	VAR robtarget OpenholeUD_1373 := [[450.39, 0.9, 181.06], [-0.062156, 0.70437, 0.703684, -0.06949], [0,0,0,0], [9E9, 9E9, 9E9, 9E9, 9E9, 9E9]];
	VAR robtarget OpenholeUD_1374 := [[446.46, 0.9, 181.82], [-0.075448, 0.70307, 0.704874, -0.056152], [0,0,0,0], [9E9, 9E9, 9E9, 9E9, 9E9, 9E9]];
	VAR robtarget OpenholeUD_1375 := [[442.53, 0.9, 182.57], [-0.088597, 0.701534, 0.705814, -0.042733], [0,0,0,0], [9E9, 9E9, 9E9, 9E9, 9E9, 9E9]];
	VAR robtarget OpenholeUD_1376 := [[438.6, 0.9, 183.32], [-0.101564, 0.699775, 0.7065, -0.029277], [0,0,0,0], [9E9, 9E9, 9E9, 9E9, 9E9, 9E9]];
	VAR robtarget OpenholeUD_1377 := [[434.67, 0.9, 184.08], [-0.114312, 0.697806, 0.70693, -0.015828], [0,0,0,0], [9E9, 9E9, 9E9, 9E9, 9E9, 9E9]];
	VAR robtarget OpenholeUD_1378 := [[430.74, 0.9, 184.83], [-0.126806, 0.695644, 0.707103, -0.002428], [0,0,0,0], [9E9, 9E9, 9E9, 9E9, 9E9, 9E9]];
	VAR robtarget OpenholeUD_1379 := [[426.82, 0.9, 185.59], [-0.139016, 0.693307, 0.707023, 0.010881], [0,0,0,0], [9E9, 9E9, 9E9, 9E9, 9E9, 9E9]];
	VAR robtarget OpenholeUD_1380 := [[422.89, 0.9, 186.34], [-0.150917, 0.690814, 0.706697, 0.024059], [0,0,0,0], [9E9, 9E9, 9E9, 9E9, 9E9, 9E9]];
	VAR robtarget OpenholeUD_1381 := [[418.96, 0.9, 187.09], [-0.162486, 0.688185, 0.706134, 0.03707], [0,0,0,0], [9E9, 9E9, 9E9, 9E9, 9E9, 9E9]];
	VAR robtarget OpenholeUD_1382 := [[415.03, 0.9, 187.85], [-0.173706, 0.685439, 0.705345, 0.049878], [0,0,0,0], [9E9, 9E9, 9E9, 9E9, 9E9, 9E9]];
	VAR robtarget OpenholeUD_1383 := [[411.1, 0.9, 188.6], [-0.184564, 0.682595, 0.704343, 0.062455], [0,0,0,0], [9E9, 9E9, 9E9, 9E9, 9E9, 9E9]];
	VAR robtarget OpenholeUD_1384 := [[407.17, 0.9, 189.35], [-0.195051, 0.679673, 0.703142, 0.074774], [0,0,0,0], [9E9, 9E9, 9E9, 9E9, 9E9, 9E9]];
	VAR robtarget OpenholeUD_1385 := [[403.25, 0.9, 190.11], [-0.205161, 0.67669, 0.701758, 0.086812], [0,0,0,0], [9E9, 9E9, 9E9, 9E9, 9E9, 9E9]];
	VAR robtarget OpenholeUD_1386 := [[399.32, 0.9, 190.86], [-0.214892, 0.673663, 0.700205, 0.098551], [0,0,0,0], [9E9, 9E9, 9E9, 9E9, 9E9, 9E9]];
	VAR robtarget OpenholeUD_1387 := [[395.39, 0.9, 191.62], [-0.224244, 0.670608, 0.698502, 0.109975], [0,0,0,0], [9E9, 9E9, 9E9, 9E9, 9E9, 9E9]];
	VAR robtarget OpenholeUD_1388 := [[389.38, 0.9, 192.77], [-0.237824, 0.665913, 0.695643, 0.126812], [0,0,0,0], [9E9, 9E9, 9E9, 9E9, 9E9, 9E9]];
	VAR robtarget OpenholeUD_1389 := [[385.38, 0.9, 192.78], [-0.183051, 0.683002, 0.683002, 0.183051], [0,0,0,0], [9E9, 9E9, 9E9, 9E9, 9E9, 9E9]];
	VAR robtarget OpenholeUD_1390 := [[381.38, 0.9, 192.79], [-0.183051, 0.683002, 0.683002, 0.183051], [0,0,0,0], [9E9, 9E9, 9E9, 9E9, 9E9, 9E9]];
	VAR robtarget OpenholeUD_1391 := [[377.38, 0.9, 192.81], [-0.183051, 0.683002, 0.683002, 0.183051], [0,0,0,0], [9E9, 9E9, 9E9, 9E9, 9E9, 9E9]];
	VAR robtarget OpenholeUD_1392 := [[373.38, 0.9, 192.82], [-0.183051, 0.683002, 0.683002, 0.183051], [0,0,0,0], [9E9, 9E9, 9E9, 9E9, 9E9, 9E9]];
	VAR robtarget OpenholeUD_1393 := [[369.38, 0.9, 192.83], [-0.183051, 0.683002, 0.683002, 0.183051], [0,0,0,0], [9E9, 9E9, 9E9, 9E9, 9E9, 9E9]];
	VAR robtarget OpenholeUD_1394 := [[369.38, 0.9, 192.83], [-0.183051, 0.683002, 0.683002, 0.183051], [0,0,0,0], [9E9, 9E9, 9E9, 9E9, 9E9, 9E9]];
	VAR robtarget OpenholeUD_1395 := [[369.38, 0.9, 192.95], [-0.183051, 0.683002, 0.683002, 0.183051], [0,0,0,0], [9E9, 9E9, 9E9, 9E9, 9E9, 9E9]];
	VAR robtarget OpenholeUD_1396 := [[373.38, 0.9, 192.94], [-0.183051, 0.683002, 0.683002, 0.183051], [0,0,0,0], [9E9, 9E9, 9E9, 9E9, 9E9, 9E9]];
	VAR robtarget OpenholeUD_1397 := [[377.38, 0.9, 192.93], [-0.183051, 0.683002, 0.683002, 0.183051], [0,0,0,0], [9E9, 9E9, 9E9, 9E9, 9E9, 9E9]];
	VAR robtarget OpenholeUD_1398 := [[381.38, 0.9, 192.91], [-0.183051, 0.683002, 0.683002, 0.183051], [0,0,0,0], [9E9, 9E9, 9E9, 9E9, 9E9, 9E9]];
	VAR robtarget OpenholeUD_1399 := [[385.38, 0.9, 192.9], [-0.183051, 0.683002, 0.683002, 0.183051], [0,0,0,0], [9E9, 9E9, 9E9, 9E9, 9E9, 9E9]];
	VAR robtarget OpenholeUD_1400 := [[389.38, 0.9, 192.89], [-0.237996, 0.665851, 0.695661, 0.126714], [0,0,0,0], [9E9, 9E9, 9E9, 9E9, 9E9, 9E9]];
	VAR robtarget OpenholeUD_1401 := [[393.31, 0.9, 192.14], [-0.229215, 0.668925, 0.697561, 0.115797], [0,0,0,0], [9E9, 9E9, 9E9, 9E9, 9E9, 9E9]];
	VAR robtarget OpenholeUD_1402 := [[397.24, 0.9, 191.38], [-0.220061, 0.671992, 0.699335, 0.10455], [0,0,0,0], [9E9, 9E9, 9E9, 9E9, 9E9, 9E9]];
	VAR robtarget OpenholeUD_1403 := [[401.17, 0.9, 190.63], [-0.210529, 0.675039, 0.700967, 0.092984], [0,0,0,0], [9E9, 9E9, 9E9, 9E9, 9E9, 9E9]];
	VAR robtarget OpenholeUD_1404 := [[405.1, 0.9, 189.87], [-0.200618, 0.678051, 0.702439, 0.08111], [0,0,0,0], [9E9, 9E9, 9E9, 9E9, 9E9, 9E9]];
	VAR robtarget OpenholeUD_1405 := [[409.02, 0.9, 189.12], [-0.190327, 0.681011, 0.703737, 0.068947], [0,0,0,0], [9E9, 9E9, 9E9, 9E9, 9E9, 9E9]];
	VAR robtarget OpenholeUD_1406 := [[412.95, 0.9, 188.37], [-0.17966, 0.683902, 0.704845, 0.056513], [0,0,0,0], [9E9, 9E9, 9E9, 9E9, 9E9, 9E9]];
	VAR robtarget OpenholeUD_1407 := [[416.88, 0.9, 187.61], [-0.168625, 0.686706, 0.705747, 0.043835], [0,0,0,0], [9E9, 9E9, 9E9, 9E9, 9E9, 9E9]];
	VAR robtarget OpenholeUD_1408 := [[420.81, 0.9, 186.86], [-0.157232, 0.689404, 0.70643, 0.030939], [0,0,0,0], [9E9, 9E9, 9E9, 9E9, 9E9, 9E9]];
	VAR robtarget OpenholeUD_1409 := [[424.74, 0.9, 186.1], [-0.145497, 0.691976, 0.706881, 0.017859], [0,0,0,0], [9E9, 9E9, 9E9, 9E9, 9E9, 9E9]];
	VAR robtarget OpenholeUD_1410 := [[428.67, 0.9, 185.35], [-0.133439, 0.694402, 0.707092, 0.004628], [0,0,0,0], [9E9, 9E9, 9E9, 9E9, 9E9, 9E9]];
	VAR robtarget OpenholeUD_1411 := [[432.59, 0.9, 184.6], [-0.121082, 0.696663, 0.707053, -0.008715], [0,0,0,0], [9E9, 9E9, 9E9, 9E9, 9E9, 9E9]];
	VAR robtarget OpenholeUD_1412 := [[436.52, 0.9, 183.84], [-0.108454, 0.69874, 0.70676, -0.02213], [0,0,0,0], [9E9, 9E9, 9E9, 9E9, 9E9, 9E9]];
	VAR robtarget OpenholeUD_1413 := [[440.45, 0.9, 183.09], [-0.095587, 0.700616, 0.706211, -0.035574], [0,0,0,0], [9E9, 9E9, 9E9, 9E9, 9E9, 9E9]];
	VAR robtarget OpenholeUD_1414 := [[444.38, 0.9, 182.33], [-0.082516, 0.702276, 0.705407, -0.049004], [0,0,0,0], [9E9, 9E9, 9E9, 9E9, 9E9, 9E9]];
	VAR robtarget OpenholeUD_1415 := [[448.31, 0.9, 181.58], [-0.069281, 0.703705, 0.70435, -0.062375], [0,0,0,0], [9E9, 9E9, 9E9, 9E9, 9E9, 9E9]];
	VAR robtarget OpenholeUD_1416 := [[452.24, 0.9, 180.83], [-0.055922, 0.704892, 0.703049, -0.075646], [0,0,0,0], [9E9, 9E9, 9E9, 9E9, 9E9, 9E9]];
	VAR robtarget OpenholeUD_1417 := [[456.16, 0.9, 180.07], [-0.042483, 0.705829, 0.701512, -0.088775], [0,0,0,0], [9E9, 9E9, 9E9, 9E9, 9E9, 9E9]];
	VAR robtarget OpenholeUD_1418 := [[460.09, 0.9, 179.32], [-0.029008, 0.706512, 0.699752, -0.101721], [0,0,0,0], [9E9, 9E9, 9E9, 9E9, 9E9, 9E9]];
	VAR robtarget OpenholeUD_1419 := [[464.02, 0.9, 178.57], [-0.01554, 0.706936, 0.697783, -0.114448], [0,0,0,0], [9E9, 9E9, 9E9, 9E9, 9E9, 9E9]];
	VAR robtarget OpenholeUD_1420 := [[467.95, 0.9, 177.81], [-0.002122, 0.707104, 0.695623, -0.126921], [0,0,0,0], [9E9, 9E9, 9E9, 9E9, 9E9, 9E9]];
	VAR robtarget OpenholeUD_1421 := [[471.88, 0.9, 177.06], [0.011202, 0.707018, 0.693288, -0.139112], [0,0,0,0], [9E9, 9E9, 9E9, 9E9, 9E9, 9E9]];
	VAR robtarget OpenholeUD_1422 := [[475.81, 0.9, 176.3], [0.024395, 0.706686, 0.690797, -0.150995], [0,0,0,0], [9E9, 9E9, 9E9, 9E9, 9E9, 9E9]];
	VAR robtarget OpenholeUD_1423 := [[479.73, 0.9, 175.55], [0.037417, 0.706116, 0.68817, -0.162547], [0,0,0,0], [9E9, 9E9, 9E9, 9E9, 9E9, 9E9]];
	VAR robtarget OpenholeUD_1424 := [[483.66, 0.9, 174.8], [0.050236, 0.70532, 0.685427, -0.173751], [0,0,0,0], [9E9, 9E9, 9E9, 9E9, 9E9, 9E9]];
	VAR robtarget OpenholeUD_1425 := [[487.59, 0.9, 174.04], [0.062822, 0.704311, 0.682587, -0.184594], [0,0,0,0], [9E9, 9E9, 9E9, 9E9, 9E9, 9E9]];
	VAR robtarget OpenholeUD_1426 := [[491.52, 0.9, 173.29], [0.075148, 0.703102, 0.679668, -0.195068], [0,0,0,0], [9E9, 9E9, 9E9, 9E9, 9E9, 9E9]];
	VAR robtarget OpenholeUD_1427 := [[495.45, 0.9, 172.53], [0.087191, 0.701711, 0.676688, -0.205165], [0,0,0,0], [9E9, 9E9, 9E9, 9E9, 9E9, 9E9]];
	VAR robtarget OpenholeUD_1428 := [[499.38, 0.9, 171.78], [0.098933, 0.700152, 0.673665, -0.214885], [0,0,0,0], [9E9, 9E9, 9E9, 9E9, 9E9, 9E9]];
	VAR robtarget OpenholeUD_1429 := [[503.3, 0.9, 171.03], [0.110359, 0.698442, 0.670613, -0.224228], [0,0,0,0], [9E9, 9E9, 9E9, 9E9, 9E9, 9E9]];
	VAR robtarget OpenholeUD_1430 := [[509.31, 0.9, 169.87], [0.183051, 0.683002, 0.683002, -0.183051], [0,0,0,0], [9E9, 9E9, 9E9, 9E9, 9E9, 9E9]];
	VAR robtarget OpenholeUD_1431 := [[513.31, 0.9, 169.86], [0.183051, 0.683002, 0.683002, -0.183051], [0,0,0,0], [9E9, 9E9, 9E9, 9E9, 9E9, 9E9]];
	VAR robtarget OpenholeUD_1432 := [[517.31, 0.9, 169.85], [0.183051, 0.683002, 0.683002, -0.183051], [0,0,0,0], [9E9, 9E9, 9E9, 9E9, 9E9, 9E9]];
	VAR robtarget OpenholeUD_1433 := [[521.31, 0.9, 169.84], [0.183051, 0.683002, 0.683002, -0.183051], [0,0,0,0], [9E9, 9E9, 9E9, 9E9, 9E9, 9E9]];
	VAR robtarget OpenholeUD_1434 := [[525.31, 0.9, 169.82], [0.183051, 0.683002, 0.683002, -0.183051], [0,0,0,0], [9E9, 9E9, 9E9, 9E9, 9E9, 9E9]];
	VAR robtarget OpenholeUD_1435 := [[529.31, 0.9, 169.81], [0.183051, 0.683002, 0.683002, -0.183051], [0,0,0,0], [9E9, 9E9, 9E9, 9E9, 9E9, 9E9]];
	VAR robtarget OpenholeUD_1436 := [[529.31, 0.9, 169.81], [0.183051, 0.683002, 0.683002, -0.183051], [0,0,0,0], [9E9, 9E9, 9E9, 9E9, 9E9, 9E9]];
	VAR robtarget OpenholeUD_1437 := [[529.31, -0.3, 170.5], [0.183051, 0.683002, 0.683002, -0.183051], [0,0,0,0], [9E9, 9E9, 9E9, 9E9, 9E9, 9E9]];
	VAR robtarget OpenholeUD_1438 := [[525.31, -0.3, 170.52], [0.183051, 0.683002, 0.683002, -0.183051], [0,0,0,0], [9E9, 9E9, 9E9, 9E9, 9E9, 9E9]];
	VAR robtarget OpenholeUD_1439 := [[521.31, -0.3, 170.53], [0.183051, 0.683002, 0.683002, -0.183051], [0,0,0,0], [9E9, 9E9, 9E9, 9E9, 9E9, 9E9]];
	VAR robtarget OpenholeUD_1440 := [[517.31, -0.3, 170.54], [0.183051, 0.683002, 0.683002, -0.183051], [0,0,0,0], [9E9, 9E9, 9E9, 9E9, 9E9, 9E9]];
	VAR robtarget OpenholeUD_1441 := [[509.31, -0.3, 170.57], [0.183051, 0.683002, 0.683002, -0.183051], [0,0,0,0], [9E9, 9E9, 9E9, 9E9, 9E9, 9E9]];
	VAR robtarget OpenholeUD_1442 := [[505.38, -0.3, 171.28], [0.119709, 0.6969, 0.670123, -0.225689], [0,0,0,0], [9E9, 9E9, 9E9, 9E9, 9E9, 9E9]];
	VAR robtarget OpenholeUD_1443 := [[501.44, -0.3, 171.99], [0.108491, 0.698734, 0.673161, -0.21646], [0,0,0,0], [9E9, 9E9, 9E9, 9E9, 9E9, 9E9]];
	VAR robtarget OpenholeUD_1444 := [[497.5, -0.3, 172.7], [0.096948, 0.700429, 0.676174, -0.206855], [0,0,0,0], [9E9, 9E9, 9E9, 9E9, 9E9, 9E9]];
	VAR robtarget OpenholeUD_1445 := [[493.57, -0.3, 173.41], [0.085091, 0.701968, 0.679147, -0.196873], [0,0,0,0], [9E9, 9E9, 9E9, 9E9, 9E9, 9E9]];
	VAR robtarget OpenholeUD_1446 := [[489.63, -0.3, 174.12], [0.072938, 0.703335, 0.682065, -0.186514], [0,0,0,0], [9E9, 9E9, 9E9, 9E9, 9E9, 9E9]];
	VAR robtarget OpenholeUD_1447 := [[485.69, -0.3, 174.83], [0.060507, 0.704513, 0.684909, -0.175783], [0,0,0,0], [9E9, 9E9, 9E9, 9E9, 9E9, 9E9]];
	VAR robtarget OpenholeUD_1448 := [[481.76, -0.3, 175.54], [0.047824, 0.705488, 0.687661, -0.164688], [0,0,0,0], [9E9, 9E9, 9E9, 9E9, 9E9, 9E9]];
	VAR robtarget OpenholeUD_1449 := [[477.82, -0.3, 176.25], [0.034916, 0.706244, 0.690303, -0.153239], [0,0,0,0], [9E9, 9E9, 9E9, 9E9, 9E9, 9E9]];
	VAR robtarget OpenholeUD_1450 := [[473.88, -0.3, 176.96], [0.021815, 0.70677, 0.692814, -0.141454], [0,0,0,0], [9E9, 9E9, 9E9, 9E9, 9E9, 9E9]];
	VAR robtarget OpenholeUD_1451 := [[469.95, -0.3, 177.67], [0.008556, 0.707055, 0.695175, -0.129352], [0,0,0,0], [9E9, 9E9, 9E9, 9E9, 9E9, 9E9]];
	VAR robtarget OpenholeUD_1452 := [[466.01, -0.3, 178.38], [-0.004823, 0.70709, 0.697367, -0.116957], [0,0,0,0], [9E9, 9E9, 9E9, 9E9, 9E9, 9E9]];
	VAR robtarget OpenholeUD_1453 := [[462.07, -0.3, 179.09], [-0.01828, 0.70687, 0.699372, -0.104298], [0,0,0,0], [9E9, 9E9, 9E9, 9E9, 9E9, 9E9]];
	VAR robtarget OpenholeUD_1454 := [[458.14, -0.3, 179.8], [-0.031774, 0.706393, 0.701174, -0.091408], [0,0,0,0], [9E9, 9E9, 9E9, 9E9, 9E9, 9E9]];
	VAR robtarget OpenholeUD_1455 := [[454.2, -0.3, 180.51], [-0.045259, 0.705657, 0.702756, -0.078321], [0,0,0,0], [9E9, 9E9, 9E9, 9E9, 9E9, 9E9]];
	VAR robtarget OpenholeUD_1456 := [[450.27, -0.3, 181.22], [-0.058693, 0.704667, 0.704106, -0.065078], [0,0,0,0], [9E9, 9E9, 9E9, 9E9, 9E9, 9E9]];
	VAR robtarget OpenholeUD_1457 := [[446.33, -0.3, 181.93], [-0.072031, 0.703428, 0.705213, -0.051719], [0,0,0,0], [9E9, 9E9, 9E9, 9E9, 9E9, 9E9]];
	VAR robtarget OpenholeUD_1458 := [[442.39, -0.3, 182.64], [-0.08523, 0.701951, 0.70607, -0.038286], [0,0,0,0], [9E9, 9E9, 9E9, 9E9, 9E9, 9E9]];
	VAR robtarget OpenholeUD_1459 := [[438.46, -0.3, 183.35], [-0.09825, 0.700248, 0.706671, -0.024825], [0,0,0,0], [9E9, 9E9, 9E9, 9E9, 9E9, 9E9]];
	VAR robtarget OpenholeUD_1460 := [[434.52, -0.3, 184.06], [-0.111054, 0.698332, 0.707015, -0.011378], [0,0,0,0], [9E9, 9E9, 9E9, 9E9, 9E9, 9E9]];
	VAR robtarget OpenholeUD_1461 := [[430.58, -0.3, 184.77], [-0.123606, 0.696219, 0.707104, 0.002011], [0,0,0,0], [9E9, 9E9, 9E9, 9E9, 9E9, 9E9]];
	VAR robtarget OpenholeUD_1462 := [[426.65, -0.3, 185.48], [-0.135877, 0.693929, 0.706941, 0.015302], [0,0,0,0], [9E9, 9E9, 9E9, 9E9, 9E9, 9E9]];
	VAR robtarget OpenholeUD_1463 := [[422.71, -0.3, 186.19], [-0.14784, 0.691479, 0.706534, 0.028455], [0,0,0,0], [9E9, 9E9, 9E9, 9E9, 9E9, 9E9]];
	VAR robtarget OpenholeUD_1464 := [[418.77, -0.3, 186.9], [-0.159473, 0.688889, 0.705892, 0.041433], [0,0,0,0], [9E9, 9E9, 9E9, 9E9, 9E9, 9E9]];
	VAR robtarget OpenholeUD_1465 := [[414.84, -0.3, 187.6], [-0.170757, 0.686179, 0.705026, 0.054203], [0,0,0,0], [9E9, 9E9, 9E9, 9E9, 9E9, 9E9]];
	VAR robtarget OpenholeUD_1466 := [[410.9, -0.3, 188.31], [-0.181679, 0.683369, 0.703951, 0.066735], [0,0,0,0], [9E9, 9E9, 9E9, 9E9, 9E9, 9E9]];
	VAR robtarget OpenholeUD_1467 := [[406.96, -0.3, 189.02], [-0.19223, 0.680476, 0.702679, 0.079005], [0,0,0,0], [9E9, 9E9, 9E9, 9E9, 9E9, 9E9]];
	VAR robtarget OpenholeUD_1468 := [[403.03, -0.3, 189.73], [-0.202403, 0.67752, 0.701228, 0.090989], [0,0,0,0], [9E9, 9E9, 9E9, 9E9, 9E9, 9E9]];
	VAR robtarget OpenholeUD_1469 := [[399.09, -0.3, 190.44], [-0.212197, 0.674516, 0.699613, 0.10267], [0,0,0,0], [9E9, 9E9, 9E9, 9E9, 9E9, 9E9]];
	VAR robtarget OpenholeUD_1470 := [[395.15, -0.3, 191.15], [-0.221612, 0.671482, 0.697851, 0.114033], [0,0,0,0], [9E9, 9E9, 9E9, 9E9, 9E9, 9E9]];
	VAR robtarget OpenholeUD_1471 := [[389.38, -0.3, 192.2], [-0.234744, 0.667005, 0.695035, 0.130104], [0,0,0,0], [9E9, 9E9, 9E9, 9E9, 9E9, 9E9]];
	VAR robtarget OpenholeUD_1472 := [[385.38, -0.3, 192.21], [-0.183051, 0.683002, 0.683002, 0.183051], [0,0,0,0], [9E9, 9E9, 9E9, 9E9, 9E9, 9E9]];
	VAR robtarget OpenholeUD_1473 := [[381.38, -0.3, 192.22], [-0.183051, 0.683002, 0.683002, 0.183051], [0,0,0,0], [9E9, 9E9, 9E9, 9E9, 9E9, 9E9]];
	VAR robtarget OpenholeUD_1474 := [[377.38, -0.3, 192.23], [-0.183051, 0.683002, 0.683002, 0.183051], [0,0,0,0], [9E9, 9E9, 9E9, 9E9, 9E9, 9E9]];
	VAR robtarget OpenholeUD_1475 := [[373.38, -0.3, 192.25], [-0.183051, 0.683002, 0.683002, 0.183051], [0,0,0,0], [9E9, 9E9, 9E9, 9E9, 9E9, 9E9]];
	VAR robtarget OpenholeUD_1476 := [[369.38, -0.3, 192.26], [-0.183051, 0.683002, 0.683002, 0.183051], [0,0,0,0], [9E9, 9E9, 9E9, 9E9, 9E9, 9E9]];
	VAR robtarget OpenholeUD_1477 := [[369.38, -0.3, 192.26], [-0.183051, 0.683002, 0.683002, 0.183051], [0,0,0,0], [9E9, 9E9, 9E9, 9E9, 9E9, 9E9]];
	VAR robtarget OpenholeUD_1478 := [[369.38, -1.5, 191.57], [-0.183051, 0.683002, 0.683002, 0.183051], [0,0,0,0], [9E9, 9E9, 9E9, 9E9, 9E9, 9E9]];
	VAR robtarget OpenholeUD_1479 := [[373.38, -1.5, 191.55], [-0.183051, 0.683002, 0.683002, 0.183051], [0,0,0,0], [9E9, 9E9, 9E9, 9E9, 9E9, 9E9]];
	VAR robtarget OpenholeUD_1480 := [[377.38, -1.5, 191.54], [-0.183051, 0.683002, 0.683002, 0.183051], [0,0,0,0], [9E9, 9E9, 9E9, 9E9, 9E9, 9E9]];
	VAR robtarget OpenholeUD_1481 := [[381.38, -1.5, 191.53], [-0.183051, 0.683002, 0.683002, 0.183051], [0,0,0,0], [9E9, 9E9, 9E9, 9E9, 9E9, 9E9]];
	VAR robtarget OpenholeUD_1482 := [[385.38, -1.5, 191.52], [-0.183051, 0.683002, 0.683002, 0.183051], [0,0,0,0], [9E9, 9E9, 9E9, 9E9, 9E9, 9E9]];
	VAR robtarget OpenholeUD_1483 := [[389.38, -1.5, 191.5], [-0.231476, 0.668146, 0.69439, 0.133501], [0,0,0,0], [9E9, 9E9, 9E9, 9E9, 9E9, 9E9]];
	VAR robtarget OpenholeUD_1484 := [[393.32, -1.5, 190.84], [-0.222527, 0.67118, 0.696386, 0.122664], [0,0,0,0], [9E9, 9E9, 9E9, 9E9, 9E9, 9E9]];
	VAR robtarget OpenholeUD_1485 := [[397.27, -1.5, 190.17], [-0.213203, 0.674199, 0.698262, 0.111491], [0,0,0,0], [9E9, 9E9, 9E9, 9E9, 9E9, 9E9]];
	VAR robtarget OpenholeUD_1486 := [[401.21, -1.5, 189.51], [-0.203502, 0.67719, 0.700001, 0.099992], [0,0,0,0], [9E9, 9E9, 9E9, 9E9, 9E9, 9E9]];
	VAR robtarget OpenholeUD_1487 := [[405.15, -1.5, 188.84], [-0.193422, 0.680138, 0.701587, 0.088179], [0,0,0,0], [9E9, 9E9, 9E9, 9E9, 9E9, 9E9]];
	VAR robtarget OpenholeUD_1488 := [[409.1, -1.5, 188.17], [-0.182963, 0.683026, 0.703003, 0.076067], [0,0,0,0], [9E9, 9E9, 9E9, 9E9, 9E9, 9E9]];
	VAR robtarget OpenholeUD_1489 := [[413.04, -1.5, 187.51], [-0.172131, 0.685836, 0.704234, 0.063677], [0,0,0,0], [9E9, 9E9, 9E9, 9E9, 9E9, 9E9]];
	VAR robtarget OpenholeUD_1490 := [[416.99, -1.5, 186.84], [-0.160934, 0.688549, 0.705263, 0.051033], [0,0,0,0], [9E9, 9E9, 9E9, 9E9, 9E9, 9E9]];
	VAR robtarget OpenholeUD_1491 := [[420.93, -1.5, 186.18], [-0.149385, 0.691147, 0.706076, 0.038161], [0,0,0,0], [9E9, 9E9, 9E9, 9E9, 9E9, 9E9]];
	VAR robtarget OpenholeUD_1492 := [[424.88, -1.5, 185.51], [-0.137499, 0.693609, 0.706661, 0.025094], [0,0,0,0], [9E9, 9E9, 9E9, 9E9, 9E9, 9E9]];
	VAR robtarget OpenholeUD_1493 := [[428.82, -1.5, 184.85], [-0.125298, 0.695917, 0.707007, 0.011865], [0,0,0,0], [9E9, 9E9, 9E9, 9E9, 9E9, 9E9]];
	VAR robtarget OpenholeUD_1494 := [[432.76, -1.5, 184.18], [-0.112808, 0.69805, 0.707105, -0.001486], [0,0,0,0], [9E9, 9E9, 9E9, 9E9, 9E9, 9E9]];
	VAR robtarget OpenholeUD_1495 := [[436.71, -1.5, 183.51], [-0.100057, 0.699992, 0.706949, -0.014921], [0,0,0,0], [9E9, 9E9, 9E9, 9E9, 9E9, 9E9]];
	VAR robtarget OpenholeUD_1496 := [[440.65, -1.5, 182.85], [-0.087079, 0.701724, 0.706536, -0.028395], [0,0,0,0], [9E9, 9E9, 9E9, 9E9, 9E9, 9E9]];
	VAR robtarget OpenholeUD_1497 := [[444.6, -1.5, 182.18], [-0.073911, 0.703233, 0.705866, -0.041866], [0,0,0,0], [9E9, 9E9, 9E9, 9E9, 9E9, 9E9]];
	VAR robtarget OpenholeUD_1498 := [[448.54, -1.5, 181.52], [-0.060592, 0.704506, 0.704942, -0.05529], [0,0,0,0], [9E9, 9E9, 9E9, 9E9, 9E9, 9E9]];
	VAR robtarget OpenholeUD_1499 := [[452.49, -1.5, 180.85], [-0.047165, 0.705532, 0.703769, -0.068623], [0,0,0,0], [9E9, 9E9, 9E9, 9E9, 9E9, 9E9]];
	VAR robtarget OpenholeUD_1500 := [[456.43, -1.5, 180.19], [-0.033673, 0.706305, 0.702357, -0.081823], [0,0,0,0], [9E9, 9E9, 9E9, 9E9, 9E9, 9E9]];
	VAR robtarget OpenholeUD_1501 := [[460.37, -1.5, 179.52], [-0.020161, 0.706819, 0.700716, -0.094849], [0,0,0,0], [9E9, 9E9, 9E9, 9E9, 9E9, 9E9]];
	VAR robtarget OpenholeUD_1502 := [[464.32, -1.5, 178.85], [-0.006672, 0.707075, 0.698862, -0.107665], [0,0,0,0], [9E9, 9E9, 9E9, 9E9, 9E9, 9E9]];
	VAR robtarget OpenholeUD_1503 := [[468.26, -1.5, 178.19], [0.006749, 0.707075, 0.69681, -0.120234], [0,0,0,0], [9E9, 9E9, 9E9, 9E9, 9E9, 9E9]];
	VAR robtarget OpenholeUD_1504 := [[472.21, -1.5, 177.52], [0.020061, 0.706822, 0.694577, -0.132527], [0,0,0,0], [9E9, 9E9, 9E9, 9E9, 9E9, 9E9]];
	VAR robtarget OpenholeUD_1505 := [[476.15, -1.5, 176.86], [0.033225, 0.706326, 0.692181, -0.144516], [0,0,0,0], [9E9, 9E9, 9E9, 9E9, 9E9, 9E9]];
	VAR robtarget OpenholeUD_1506 := [[480.09, -1.5, 176.19], [0.046205, 0.705596, 0.689643, -0.15618], [0,0,0,0], [9E9, 9E9, 9E9, 9E9, 9E9, 9E9]];
	VAR robtarget OpenholeUD_1507 := [[484.04, -1.5, 175.53], [0.058967, 0.704644, 0.686982, -0.1675], [0,0,0,0], [9E9, 9E9, 9E9, 9E9, 9E9, 9E9]];
	VAR robtarget OpenholeUD_1508 := [[487.98, -1.5, 174.86], [0.071483, 0.703484, 0.684216, -0.178463], [0,0,0,0], [9E9, 9E9, 9E9, 9E9, 9E9, 9E9]];
	VAR robtarget OpenholeUD_1509 := [[491.93, -1.5, 174.19], [0.083726, 0.702132, 0.681365, -0.189057], [0,0,0,0], [9E9, 9E9, 9E9, 9E9, 9E9, 9E9]];
	VAR robtarget OpenholeUD_1510 := [[495.87, -1.5, 173.53], [0.095676, 0.700604, 0.678446, -0.199276], [0,0,0,0], [9E9, 9E9, 9E9, 9E9, 9E9, 9E9]];
	VAR robtarget OpenholeUD_1511 := [[499.82, -1.5, 172.86], [0.107315, 0.698916, 0.675477, -0.209119], [0,0,0,0], [9E9, 9E9, 9E9, 9E9, 9E9, 9E9]];
	VAR robtarget OpenholeUD_1512 := [[503.76, -1.5, 172.2], [0.118629, 0.697085, 0.672473, -0.218585], [0,0,0,0], [9E9, 9E9, 9E9, 9E9, 9E9, 9E9]];
	VAR robtarget OpenholeUD_1513 := [[509.31, -1.5, 171.26], [0.183051, 0.683002, 0.683002, -0.183051], [0,0,0,0], [9E9, 9E9, 9E9, 9E9, 9E9, 9E9]];
	VAR robtarget OpenholeUD_1514 := [[513.31, -1.5, 171.25], [0.183051, 0.683002, 0.683002, -0.183051], [0,0,0,0], [9E9, 9E9, 9E9, 9E9, 9E9, 9E9]];
	VAR robtarget OpenholeUD_1515 := [[517.31, -1.5, 171.23], [0.183051, 0.683002, 0.683002, -0.183051], [0,0,0,0], [9E9, 9E9, 9E9, 9E9, 9E9, 9E9]];
	VAR robtarget OpenholeUD_1516 := [[521.31, -1.5, 171.22], [0.183051, 0.683002, 0.683002, -0.183051], [0,0,0,0], [9E9, 9E9, 9E9, 9E9, 9E9, 9E9]];
	VAR robtarget OpenholeUD_1517 := [[525.31, -1.5, 171.21], [0.183051, 0.683002, 0.683002, -0.183051], [0,0,0,0], [9E9, 9E9, 9E9, 9E9, 9E9, 9E9]];
	VAR robtarget OpenholeUD_1518 := [[529.31, -1.5, 171.2], [0.183051, 0.683002, 0.683002, -0.183051], [0,0,0,0], [9E9, 9E9, 9E9, 9E9, 9E9, 9E9]];
	VAR robtarget OpenholeUD_1519 := [[529.31, -1.5, 171.2], [0.183051, 0.683002, 0.683002, -0.183051], [0,0,0,0], [9E9, 9E9, 9E9, 9E9, 9E9, 9E9]];
	VAR robtarget OpenholeUD_1520 := [[529.32, -2.7, 171.89], [0.183051, 0.683002, 0.683002, -0.183051], [0,0,0,0], [9E9, 9E9, 9E9, 9E9, 9E9, 9E9]];
	VAR robtarget OpenholeUD_1521 := [[525.32, -2.7, 171.9], [0.183051, 0.683002, 0.683002, -0.183051], [0,0,0,0], [9E9, 9E9, 9E9, 9E9, 9E9, 9E9]];
	VAR robtarget OpenholeUD_1522 := [[521.32, -2.7, 171.92], [0.183051, 0.683002, 0.683002, -0.183051], [0,0,0,0], [9E9, 9E9, 9E9, 9E9, 9E9, 9E9]];
	VAR robtarget OpenholeUD_1523 := [[517.32, -2.7, 171.93], [0.183051, 0.683002, 0.683002, -0.183051], [0,0,0,0], [9E9, 9E9, 9E9, 9E9, 9E9, 9E9]];
	VAR robtarget OpenholeUD_1524 := [[513.32, -2.7, 171.94], [0.183051, 0.683002, 0.683002, -0.183051], [0,0,0,0], [9E9, 9E9, 9E9, 9E9, 9E9, 9E9]];
	VAR robtarget OpenholeUD_1525 := [[509.32, -2.7, 171.95], [0.183051, 0.683002, 0.683002, -0.183051], [0,0,0,0], [9E9, 9E9, 9E9, 9E9, 9E9, 9E9]];
	VAR robtarget OpenholeUD_1526 := [[505.37, -2.7, 172.57], [0.126607, 0.69568, 0.672344, -0.218982], [0,0,0,0], [9E9, 9E9, 9E9, 9E9, 9E9, 9E9]];
	VAR robtarget OpenholeUD_1527 := [[501.41, -2.7, 173.2], [0.115469, 0.697615, 0.675332, -0.209586], [0,0,0,0], [9E9, 9E9, 9E9, 9E9, 9E9, 9E9]];
	VAR robtarget OpenholeUD_1528 := [[497.46, -2.7, 173.82], [0.103999, 0.699417, 0.678288, -0.199814], [0,0,0,0], [9E9, 9E9, 9E9, 9E9, 9E9, 9E9]];
	VAR robtarget OpenholeUD_1529 := [[493.51, -2.7, 174.44], [0.092208, 0.701069, 0.681195, -0.189665], [0,0,0,0], [9E9, 9E9, 9E9, 9E9, 9E9, 9E9]];
	VAR robtarget OpenholeUD_1530 := [[489.56, -2.7, 175.06], [0.080112, 0.702554, 0.684038, -0.179141], [0,0,0,0], [9E9, 9E9, 9E9, 9E9, 9E9, 9E9]];
	VAR robtarget OpenholeUD_1531 := [[485.61, -2.7, 175.68], [0.067731, 0.703855, 0.686799, -0.168247], [0,0,0,0], [9E9, 9E9, 9E9, 9E9, 9E9, 9E9]];
	VAR robtarget OpenholeUD_1532 := [[481.66, -2.7, 176.3], [0.055087, 0.704958, 0.689459, -0.156993], [0,0,0,0], [9E9, 9E9, 9E9, 9E9, 9E9, 9E9]];
	VAR robtarget OpenholeUD_1533 := [[477.71, -2.7, 176.92], [0.042209, 0.705846, 0.691998, -0.145392], [0,0,0,0], [9E9, 9E9, 9E9, 9E9, 9E9, 9E9]];
	VAR robtarget OpenholeUD_1534 := [[473.75, -2.7, 177.54], [0.029126, 0.706507, 0.694398, -0.133461], [0,0,0,0], [9E9, 9E9, 9E9, 9E9, 9E9, 9E9]];
	VAR robtarget OpenholeUD_1535 := [[469.8, -2.7, 178.17], [0.015875, 0.706929, 0.696639, -0.121221], [0,0,0,0], [9E9, 9E9, 9E9, 9E9, 9E9, 9E9]];
	VAR robtarget OpenholeUD_1536 := [[465.85, -2.7, 178.79], [0.002493, 0.707102, 0.698702, -0.108697], [0,0,0,0], [9E9, 9E9, 9E9, 9E9, 9E9, 9E9]];
	VAR robtarget OpenholeUD_1537 := [[461.9, -2.7, 179.41], [-0.01098, 0.707022, 0.700571, -0.095921], [0,0,0,0], [9E9, 9E9, 9E9, 9E9, 9E9, 9E9]];
	VAR robtarget OpenholeUD_1538 := [[457.95, -2.7, 180.03], [-0.0245, 0.706682, 0.702228, -0.082925], [0,0,0,0], [9E9, 9E9, 9E9, 9E9, 9E9, 9E9]];
	VAR robtarget OpenholeUD_1539 := [[454, -2.7, 180.65], [-0.038024, 0.706084, 0.703659, -0.069746], [0,0,0,0], [9E9, 9E9, 9E9, 9E9, 9E9, 9E9]];
	VAR robtarget OpenholeUD_1540 := [[450.05, -2.7, 181.27], [-0.051507, 0.705228, 0.704852, -0.056424], [0,0,0,0], [9E9, 9E9, 9E9, 9E9, 9E9, 9E9]];
	VAR robtarget OpenholeUD_1541 := [[446.09, -2.7, 181.89], [-0.064904, 0.704122, 0.705798, -0.043002], [0,0,0,0], [9E9, 9E9, 9E9, 9E9, 9E9, 9E9]];
	VAR robtarget OpenholeUD_1542 := [[442.14, -2.7, 182.51], [-0.078173, 0.702772, 0.70649, -0.029522], [0,0,0,0], [9E9, 9E9, 9E9, 9E9, 9E9, 9E9]];
	VAR robtarget OpenholeUD_1543 := [[438.19, -2.7, 183.14], [-0.091273, 0.701191, 0.706925, -0.01603], [0,0,0,0], [9E9, 9E9, 9E9, 9E9, 9E9, 9E9]];
	VAR robtarget OpenholeUD_1544 := [[434.24, -2.7, 183.76], [-0.104164, 0.699392, 0.707102, -0.002568], [0,0,0,0], [9E9, 9E9, 9E9, 9E9, 9E9, 9E9]];
	VAR robtarget OpenholeUD_1545 := [[430.29, -2.7, 184.38], [-0.116812, 0.697392, 0.707024, 0.010821], [0,0,0,0], [9E9, 9E9, 9E9, 9E9, 9E9, 9E9]];
	VAR robtarget OpenholeUD_1546 := [[426.34, -2.7, 185], [-0.129185, 0.695206, 0.706696, 0.024094], [0,0,0,0], [9E9, 9E9, 9E9, 9E9, 9E9, 9E9]];
	VAR robtarget OpenholeUD_1547 := [[422.38, -2.7, 185.62], [-0.141256, 0.692854, 0.706127, 0.037214], [0,0,0,0], [9E9, 9E9, 9E9, 9E9, 9E9, 9E9]];
	VAR robtarget OpenholeUD_1548 := [[418.43, -2.7, 186.24], [-0.153002, 0.690355, 0.705326, 0.050145], [0,0,0,0], [9E9, 9E9, 9E9, 9E9, 9E9, 9E9]];
	VAR robtarget OpenholeUD_1549 := [[414.48, -2.7, 186.86], [-0.164403, 0.687729, 0.704308, 0.062855], [0,0,0,0], [9E9, 9E9, 9E9, 9E9, 9E9, 9E9]];
	VAR robtarget OpenholeUD_1550 := [[410.53, -2.7, 187.48], [-0.175446, 0.684995, 0.703084, 0.075314], [0,0,0,0], [9E9, 9E9, 9E9, 9E9, 9E9, 9E9]];
	VAR robtarget OpenholeUD_1551 := [[406.58, -2.7, 188.11], [-0.186119, 0.682173, 0.701672, 0.087498], [0,0,0,0], [9E9, 9E9, 9E9, 9E9, 9E9, 9E9]];
	VAR robtarget OpenholeUD_1552 := [[402.63, -2.7, 188.73], [-0.196417, 0.679279, 0.700087, 0.099387], [0,0,0,0], [9E9, 9E9, 9E9, 9E9, 9E9, 9E9]];
	VAR robtarget OpenholeUD_1553 := [[398.68, -2.7, 189.35], [-0.206336, 0.676332, 0.698346, 0.110962], [0,0,0,0], [9E9, 9E9, 9E9, 9E9, 9E9, 9E9]];
	VAR robtarget OpenholeUD_1554 := [[394.72, -2.7, 189.97], [-0.215877, 0.673348, 0.696465, 0.122212], [0,0,0,0], [9E9, 9E9, 9E9, 9E9, 9E9, 9E9]];
	VAR robtarget OpenholeUD_1555 := [[389.38, -2.7, 190.81], [-0.228193, 0.669274, 0.693727, 0.136905], [0,0,0,0], [9E9, 9E9, 9E9, 9E9, 9E9, 9E9]];
	VAR robtarget OpenholeUD_1556 := [[385.38, -2.7, 190.82], [-0.183051, 0.683002, 0.683002, 0.183051], [0,0,0,0], [9E9, 9E9, 9E9, 9E9, 9E9, 9E9]];
	VAR robtarget OpenholeUD_1557 := [[381.38, -2.7, 190.84], [-0.183051, 0.683002, 0.683002, 0.183051], [0,0,0,0], [9E9, 9E9, 9E9, 9E9, 9E9, 9E9]];
	VAR robtarget OpenholeUD_1558 := [[377.38, -2.7, 190.85], [-0.183051, 0.683002, 0.683002, 0.183051], [0,0,0,0], [9E9, 9E9, 9E9, 9E9, 9E9, 9E9]];
	VAR robtarget OpenholeUD_1559 := [[373.38, -2.7, 190.86], [-0.183051, 0.683002, 0.683002, 0.183051], [0,0,0,0], [9E9, 9E9, 9E9, 9E9, 9E9, 9E9]];
	VAR robtarget OpenholeUD_1560 := [[369.38, -2.7, 190.87], [-0.183051, 0.683002, 0.683002, 0.183051], [0,0,0,0], [9E9, 9E9, 9E9, 9E9, 9E9, 9E9]];
	VAR robtarget OpenholeUD_1561 := [[369.38, -2.7, 190.87], [-0.183051, 0.683002, 0.683002, 0.183051], [0,0,0,0], [9E9, 9E9, 9E9, 9E9, 9E9, 9E9]];
	VAR robtarget OpenholeUD_1562 := [[369.37, -3.9, 190.18], [-0.183051, 0.683002, 0.683002, 0.183051], [0,0,0,0], [9E9, 9E9, 9E9, 9E9, 9E9, 9E9]];
	VAR robtarget OpenholeUD_1563 := [[373.37, -3.9, 190.17], [-0.183051, 0.683002, 0.683002, 0.183051], [0,0,0,0], [9E9, 9E9, 9E9, 9E9, 9E9, 9E9]];
	VAR robtarget OpenholeUD_1564 := [[377.37, -3.9, 190.15], [-0.183051, 0.683002, 0.683002, 0.183051], [0,0,0,0], [9E9, 9E9, 9E9, 9E9, 9E9, 9E9]];
	VAR robtarget OpenholeUD_1565 := [[381.37, -3.9, 190.14], [-0.183051, 0.683002, 0.683002, 0.183051], [0,0,0,0], [9E9, 9E9, 9E9, 9E9, 9E9, 9E9]];
	VAR robtarget OpenholeUD_1566 := [[385.37, -3.9, 190.13], [-0.183051, 0.683002, 0.683002, 0.183051], [0,0,0,0], [9E9, 9E9, 9E9, 9E9, 9E9, 9E9]];
	VAR robtarget OpenholeUD_1567 := [[389.37, -3.9, 190.12], [-0.224896, 0.670389, 0.693045, 0.140314], [0,0,0,0], [9E9, 9E9, 9E9, 9E9, 9E9, 9E9]];
	VAR robtarget OpenholeUD_1568 := [[393.33, -3.9, 189.54], [-0.215781, 0.673379, 0.695135, 0.129566], [0,0,0,0], [9E9, 9E9, 9E9, 9E9, 9E9, 9E9]];
	VAR robtarget OpenholeUD_1569 := [[397.29, -3.9, 188.96], [-0.206291, 0.676346, 0.697111, 0.118476], [0,0,0,0], [9E9, 9E9, 9E9, 9E9, 9E9, 9E9]];
	VAR robtarget OpenholeUD_1570 := [[401.25, -3.9, 188.39], [-0.196422, 0.679278, 0.698956, 0.107054], [0,0,0,0], [9E9, 9E9, 9E9, 9E9, 9E9, 9E9]];
	VAR robtarget OpenholeUD_1571 := [[405.21, -3.9, 187.81], [-0.186176, 0.682157, 0.700654, 0.095311], [0,0,0,0], [9E9, 9E9, 9E9, 9E9, 9E9, 9E9]];
	VAR robtarget OpenholeUD_1572 := [[409.16, -3.9, 187.23], [-0.175553, 0.684968, 0.702188, 0.083261], [0,0,0,0], [9E9, 9E9, 9E9, 9E9, 9E9, 9E9]];
	VAR robtarget OpenholeUD_1573 := [[413.12, -3.9, 186.66], [-0.16456, 0.687692, 0.703541, 0.070924], [0,0,0,0], [9E9, 9E9, 9E9, 9E9, 9E9, 9E9]];
	VAR robtarget OpenholeUD_1574 := [[417.08, -3.9, 186.08], [-0.153206, 0.69031, 0.704697, 0.058324], [0,0,0,0], [9E9, 9E9, 9E9, 9E9, 9E9, 9E9]];
	VAR robtarget OpenholeUD_1575 := [[421.04, -3.9, 185.5], [-0.141506, 0.692803, 0.705642, 0.045486], [0,0,0,0], [9E9, 9E9, 9E9, 9E9, 9E9, 9E9]];
	VAR robtarget OpenholeUD_1576 := [[425, -3.9, 184.93], [-0.129476, 0.695152, 0.706362, 0.032441], [0,0,0,0], [9E9, 9E9, 9E9, 9E9, 9E9, 9E9]];
	VAR robtarget OpenholeUD_1577 := [[428.96, -3.9, 184.35], [-0.11714, 0.697336, 0.706845, 0.019225], [0,0,0,0], [9E9, 9E9, 9E9, 9E9, 9E9, 9E9]];
	VAR robtarget OpenholeUD_1578 := [[432.91, -3.9, 183.77], [-0.104524, 0.699339, 0.707082, 0.005874], [0,0,0,0], [9E9, 9E9, 9E9, 9E9, 9E9, 9E9]];
	VAR robtarget OpenholeUD_1579 := [[436.87, -3.9, 183.2], [-0.091659, 0.701141, 0.707066, -0.007571], [0,0,0,0], [9E9, 9E9, 9E9, 9E9, 9E9, 9E9]];
	VAR robtarget OpenholeUD_1580 := [[440.83, -3.9, 182.62], [-0.078579, 0.702727, 0.706793, -0.021069], [0,0,0,0], [9E9, 9E9, 9E9, 9E9, 9E9, 9E9]];
	VAR robtarget OpenholeUD_1581 := [[444.79, -3.9, 182.05], [-0.065323, 0.704083, 0.706261, -0.034574], [0,0,0,0], [9E9, 9E9, 9E9, 9E9, 9E9, 9E9]];
	VAR robtarget OpenholeUD_1582 := [[448.75, -3.9, 181.47], [-0.05193, 0.705197, 0.705473, -0.048044], [0,0,0,0], [9E9, 9E9, 9E9, 9E9, 9E9, 9E9]];
	VAR robtarget OpenholeUD_1583 := [[452.71, -3.9, 180.89], [-0.038445, 0.706061, 0.704433, -0.061433], [0,0,0,0], [9E9, 9E9, 9E9, 9E9, 9E9, 9E9]];
	VAR robtarget OpenholeUD_1584 := [[456.66, -3.9, 180.32], [-0.024911, 0.706668, 0.70315, -0.0747], [0,0,0,0], [9E9, 9E9, 9E9, 9E9, 9E9, 9E9]];
	VAR robtarget OpenholeUD_1585 := [[460.62, -3.9, 179.74], [-0.011373, 0.707015, 0.701634, -0.087803], [0,0,0,0], [9E9, 9E9, 9E9, 9E9, 9E9, 9E9]];
	VAR robtarget OpenholeUD_1586 := [[464.58, -3.9, 179.16], [0.002125, 0.707104, 0.699899, -0.100704], [0,0,0,0], [9E9, 9E9, 9E9, 9E9, 9E9, 9E9]];
	VAR robtarget OpenholeUD_1587 := [[468.54, -3.9, 178.59], [0.01554, 0.706936, 0.69796, -0.113367], [0,0,0,0], [9E9, 9E9, 9E9, 9E9, 9E9, 9E9]];
	VAR robtarget OpenholeUD_1588 := [[472.5, -3.9, 178.01], [0.028829, 0.706519, 0.695834, -0.12576], [0,0,0,0], [9E9, 9E9, 9E9, 9E9, 9E9, 9E9]];
	VAR robtarget OpenholeUD_1589 := [[476.45, -3.9, 177.43], [0.041955, 0.705861, 0.693538, -0.137857], [0,0,0,0], [9E9, 9E9, 9E9, 9E9, 9E9, 9E9]];
	VAR robtarget OpenholeUD_1590 := [[480.41, -3.9, 176.86], [0.054882, 0.704974, 0.691093, -0.149634], [0,0,0,0], [9E9, 9E9, 9E9, 9E9, 9E9, 9E9]];
	VAR robtarget OpenholeUD_1591 := [[484.37, -3.9, 176.28], [0.067578, 0.70387, 0.688517, -0.161071], [0,0,0,0], [9E9, 9E9, 9E9, 9E9, 9E9, 9E9]];
	VAR robtarget OpenholeUD_1592 := [[488.33, -3.9, 175.7], [0.080015, 0.702565, 0.68583, -0.172153], [0,0,0,0], [9E9, 9E9, 9E9, 9E9, 9E9, 9E9]];
	VAR robtarget OpenholeUD_1593 := [[492.29, -3.9, 175.13], [0.092168, 0.701074, 0.683051, -0.18287], [0,0,0,0], [9E9, 9E9, 9E9, 9E9, 9E9, 9E9]];
	VAR robtarget OpenholeUD_1594 := [[496.25, -3.9, 174.55], [0.104017, 0.699414, 0.680197, -0.193215], [0,0,0,0], [9E9, 9E9, 9E9, 9E9, 9E9, 9E9]];
	VAR robtarget OpenholeUD_1595 := [[500.2, -3.9, 173.97], [0.115546, 0.697602, 0.677286, -0.203184], [0,0,0,0], [9E9, 9E9, 9E9, 9E9, 9E9, 9E9]];
	VAR robtarget OpenholeUD_1596 := [[504.16, -3.9, 173.4], [0.126744, 0.695655, 0.674334, -0.212777], [0,0,0,0], [9E9, 9E9, 9E9, 9E9, 9E9, 9E9]];
	VAR robtarget OpenholeUD_1597 := [[509.32, -3.9, 172.65], [0.183051, 0.683002, 0.683002, -0.183051], [0,0,0,0], [9E9, 9E9, 9E9, 9E9, 9E9, 9E9]];
	VAR robtarget OpenholeUD_1598 := [[513.32, -3.9, 172.63], [0.183051, 0.683002, 0.683002, -0.183051], [0,0,0,0], [9E9, 9E9, 9E9, 9E9, 9E9, 9E9]];
	VAR robtarget OpenholeUD_1599 := [[517.32, -3.9, 172.62], [0.183051, 0.683002, 0.683002, -0.183051], [0,0,0,0], [9E9, 9E9, 9E9, 9E9, 9E9, 9E9]];
	VAR robtarget OpenholeUD_1600 := [[521.32, -3.9, 172.61], [0.183051, 0.683002, 0.683002, -0.183051], [0,0,0,0], [9E9, 9E9, 9E9, 9E9, 9E9, 9E9]];
	VAR robtarget OpenholeUD_1601 := [[525.32, -3.9, 172.6], [0.183051, 0.683002, 0.683002, -0.183051], [0,0,0,0], [9E9, 9E9, 9E9, 9E9, 9E9, 9E9]];
	VAR robtarget OpenholeUD_1602 := [[529.32, -3.9, 172.58], [0.183051, 0.683002, 0.683002, -0.183051], [0,0,0,0], [9E9, 9E9, 9E9, 9E9, 9E9, 9E9]];
	VAR robtarget OpenholeUD_1603 := [[529.32, -3.9, 172.58], [0.183051, 0.683002, 0.683002, -0.183051], [0,0,0,0], [9E9, 9E9, 9E9, 9E9, 9E9, 9E9]];
	VAR robtarget OpenholeUD_1604 := [[529.32, -5.1, 173.28], [0.183051, 0.683002, 0.683002, -0.183051], [0,0,0,0], [9E9, 9E9, 9E9, 9E9, 9E9, 9E9]];
	VAR robtarget OpenholeUD_1605 := [[525.32, -5.1, 173.29], [0.183051, 0.683002, 0.683002, -0.183051], [0,0,0,0], [9E9, 9E9, 9E9, 9E9, 9E9, 9E9]];
	VAR robtarget OpenholeUD_1606 := [[521.32, -5.1, 173.3], [0.183051, 0.683002, 0.683002, -0.183051], [0,0,0,0], [9E9, 9E9, 9E9, 9E9, 9E9, 9E9]];
	VAR robtarget OpenholeUD_1607 := [[517.32, -5.1, 173.31], [0.183051, 0.683002, 0.683002, -0.183051], [0,0,0,0], [9E9, 9E9, 9E9, 9E9, 9E9, 9E9]];
	VAR robtarget OpenholeUD_1608 := [[513.32, -5.1, 173.33], [0.183051, 0.683002, 0.683002, -0.183051], [0,0,0,0], [9E9, 9E9, 9E9, 9E9, 9E9, 9E9]];
	VAR robtarget OpenholeUD_1609 := [[509.32, -5.1, 173.34], [0.183051, 0.683002, 0.683002, -0.183051], [0,0,0,0], [9E9, 9E9, 9E9, 9E9, 9E9, 9E9]];
	VAR robtarget OpenholeUD_1610 := [[505.36, -5.1, 173.87], [0.133535, 0.694383, 0.674509, -0.212222], [0,0,0,0], [9E9, 9E9, 9E9, 9E9, 9E9, 9E9]];
	VAR robtarget OpenholeUD_1611 := [[501.39, -5.1, 174.4], [0.122486, 0.696417, 0.677443, -0.20266], [0,0,0,0], [9E9, 9E9, 9E9, 9E9, 9E9, 9E9]];
	VAR robtarget OpenholeUD_1612 := [[497.43, -5.1, 174.93], [0.111099, 0.698324, 0.680336, -0.192723], [0,0,0,0], [9E9, 9E9, 9E9, 9E9, 9E9, 9E9]];
	VAR robtarget OpenholeUD_1613 := [[493.46, -5.1, 175.47], [0.099384, 0.700088, 0.683174, -0.182411], [0,0,0,0], [9E9, 9E9, 9E9, 9E9, 9E9, 9E9]];
	VAR robtarget OpenholeUD_1614 := [[489.5, -5.1, 176], [0.087356, 0.70169, 0.685938, -0.171726], [0,0,0,0], [9E9, 9E9, 9E9, 9E9, 9E9, 9E9]];
	VAR robtarget OpenholeUD_1615 := [[485.53, -5.1, 176.53], [0.075034, 0.703114, 0.68861, -0.160675], [0,0,0,0], [9E9, 9E9, 9E9, 9E9, 9E9, 9E9]];
	VAR robtarget OpenholeUD_1616 := [[481.57, -5.1, 177.06], [0.06244, 0.704345, 0.691172, -0.149268], [0,0,0,0], [9E9, 9E9, 9E9, 9E9, 9E9, 9E9]];
	VAR robtarget OpenholeUD_1617 := [[477.61, -5.1, 177.59], [0.049601, 0.705365, 0.693605, -0.13752], [0,0,0,0], [9E9, 9E9, 9E9, 9E9, 9E9, 9E9]];
	VAR robtarget OpenholeUD_1618 := [[473.64, -5.1, 178.12], [0.036547, 0.706162, 0.69589, -0.125449], [0,0,0,0], [9E9, 9E9, 9E9, 9E9, 9E9, 9E9]];
	VAR robtarget OpenholeUD_1619 := [[469.68, -5.1, 178.66], [0.023313, 0.706722, 0.698007, -0.113078], [0,0,0,0], [9E9, 9E9, 9E9, 9E9, 9E9, 9E9]];
	VAR robtarget OpenholeUD_1620 := [[465.71, -5.1, 179.19], [0.009936, 0.707037, 0.699938, -0.100434], [0,0,0,0], [9E9, 9E9, 9E9, 9E9, 9E9, 9E9]];
	VAR robtarget OpenholeUD_1621 := [[461.75, -5.1, 179.72], [-0.003543, 0.707098, 0.701666, -0.087548], [0,0,0,0], [9E9, 9E9, 9E9, 9E9, 9E9, 9E9]];
	VAR robtarget OpenholeUD_1622 := [[457.78, -5.1, 180.25], [-0.017082, 0.7069, 0.703176, -0.074455], [0,0,0,0], [9E9, 9E9, 9E9, 9E9, 9E9, 9E9]];
	VAR robtarget OpenholeUD_1623 := [[453.82, -5.1, 180.78], [-0.030637, 0.706443, 0.704454, -0.061194], [0,0,0,0], [9E9, 9E9, 9E9, 9E9, 9E9, 9E9]];
	VAR robtarget OpenholeUD_1624 := [[449.85, -5.1, 181.31], [-0.044162, 0.705726, 0.705489, -0.047804], [0,0,0,0], [9E9, 9E9, 9E9, 9E9, 9E9, 9E9]];
	VAR robtarget OpenholeUD_1625 := [[445.89, -5.1, 181.85], [-0.057613, 0.704756, 0.706273, -0.034329], [0,0,0,0], [9E9, 9E9, 9E9, 9E9, 9E9, 9E9]];
	VAR robtarget OpenholeUD_1626 := [[441.92, -5.1, 182.38], [-0.070947, 0.703539, 0.7068, -0.020812], [0,0,0,0], [9E9, 9E9, 9E9, 9E9, 9E9, 9E9]];
	VAR robtarget OpenholeUD_1627 := [[437.96, -5.1, 182.91], [-0.084122, 0.702085, 0.707069, -0.007299], [0,0,0,0], [9E9, 9E9, 9E9, 9E9, 9E9, 9E9]];
	VAR robtarget OpenholeUD_1628 := [[434, -5.1, 183.44], [-0.097098, 0.700408, 0.70708, 0.006167], [0,0,0,0], [9E9, 9E9, 9E9, 9E9, 9E9, 9E9]];
	VAR robtarget OpenholeUD_1629 := [[430.03, -5.1, 183.97], [-0.109839, 0.698524, 0.706837, 0.019544], [0,0,0,0], [9E9, 9E9, 9E9, 9E9, 9E9, 9E9]];
	VAR robtarget OpenholeUD_1630 := [[426.07, -5.1, 184.5], [-0.122313, 0.696448, 0.706346, 0.032791], [0,0,0,0], [9E9, 9E9, 9E9, 9E9, 9E9, 9E9]];
	VAR robtarget OpenholeUD_1631 := [[422.1, -5.1, 185.03], [-0.134491, 0.694199, 0.705617, 0.045869], [0,0,0,0], [9E9, 9E9, 9E9, 9E9, 9E9, 9E9]];
	VAR robtarget OpenholeUD_1632 := [[418.14, -5.1, 185.57], [-0.14635, 0.691796, 0.704662, 0.058743], [0,0,0,0], [9E9, 9E9, 9E9, 9E9, 9E9, 9E9]];
	VAR robtarget OpenholeUD_1633 := [[414.17, -5.1, 186.1], [-0.157869, 0.689258, 0.703494, 0.071383], [0,0,0,0], [9E9, 9E9, 9E9, 9E9, 9E9, 9E9]];
	VAR robtarget OpenholeUD_1634 := [[410.21, -5.1, 186.63], [-0.169034, 0.686606, 0.702128, 0.083761], [0,0,0,0], [9E9, 9E9, 9E9, 9E9, 9E9, 9E9]];
	VAR robtarget OpenholeUD_1635 := [[406.24, -5.1, 187.16], [-0.179832, 0.683857, 0.70058, 0.095852], [0,0,0,0], [9E9, 9E9, 9E9, 9E9, 9E9, 9E9]];
	VAR robtarget OpenholeUD_1636 := [[402.28, -5.1, 187.69], [-0.190257, 0.68103, 0.698866, 0.107638], [0,0,0,0], [9E9, 9E9, 9E9, 9E9, 9E9, 9E9]];
	VAR robtarget OpenholeUD_1637 := [[398.32, -5.1, 188.22], [-0.200304, 0.678143, 0.697004, 0.119103], [0,0,0,0], [9E9, 9E9, 9E9, 9E9, 9E9, 9E9]];
	VAR robtarget OpenholeUD_1638 := [[394.35, -5.1, 188.76], [-0.209974, 0.675212, 0.69501, 0.130234], [0,0,0,0], [9E9, 9E9, 9E9, 9E9, 9E9, 9E9]];
	VAR robtarget OpenholeUD_1639 := [[389.37, -5.1, 189.42], [-0.221586, 0.671491, 0.692345, 0.143729], [0,0,0,0], [9E9, 9E9, 9E9, 9E9, 9E9, 9E9]];
	VAR robtarget OpenholeUD_1640 := [[385.37, -5.1, 189.44], [-0.183051, 0.683002, 0.683002, 0.183051], [0,0,0,0], [9E9, 9E9, 9E9, 9E9, 9E9, 9E9]];
	VAR robtarget OpenholeUD_1641 := [[381.37, -5.1, 189.45], [-0.183051, 0.683002, 0.683002, 0.183051], [0,0,0,0], [9E9, 9E9, 9E9, 9E9, 9E9, 9E9]];
	VAR robtarget OpenholeUD_1642 := [[377.37, -5.1, 189.46], [-0.183051, 0.683002, 0.683002, 0.183051], [0,0,0,0], [9E9, 9E9, 9E9, 9E9, 9E9, 9E9]];
	VAR robtarget OpenholeUD_1643 := [[373.37, -5.1, 189.47], [-0.183051, 0.683002, 0.683002, 0.183051], [0,0,0,0], [9E9, 9E9, 9E9, 9E9, 9E9, 9E9]];
	VAR robtarget OpenholeUD_1644 := [[369.37, -5.1, 189.49], [-0.183051, 0.683002, 0.683002, 0.183051], [0,0,0,0], [9E9, 9E9, 9E9, 9E9, 9E9, 9E9]];
	VAR robtarget OpenholeUD_1645 := [[369.37, -5.1, 189.49], [-0.183051, 0.683002, 0.683002, 0.183051], [0,0,0,0], [9E9, 9E9, 9E9, 9E9, 9E9, 9E9]];
	VAR robtarget OpenholeUD_1646 := [[369.37, -6.3, 188.79], [-0.183051, 0.683002, 0.683002, 0.183051], [0,0,0,0], [9E9, 9E9, 9E9, 9E9, 9E9, 9E9]];
	VAR robtarget OpenholeUD_1647 := [[373.37, -6.3, 188.78], [-0.183051, 0.683002, 0.683002, 0.183051], [0,0,0,0], [9E9, 9E9, 9E9, 9E9, 9E9, 9E9]];
	VAR robtarget OpenholeUD_1648 := [[377.37, -6.3, 188.77], [-0.183051, 0.683002, 0.683002, 0.183051], [0,0,0,0], [9E9, 9E9, 9E9, 9E9, 9E9, 9E9]];
	VAR robtarget OpenholeUD_1649 := [[381.37, -6.3, 188.76], [-0.183051, 0.683002, 0.683002, 0.183051], [0,0,0,0], [9E9, 9E9, 9E9, 9E9, 9E9, 9E9]];
	VAR robtarget OpenholeUD_1650 := [[385.37, -6.3, 188.74], [-0.183051, 0.683002, 0.683002, 0.183051], [0,0,0,0], [9E9, 9E9, 9E9, 9E9, 9E9, 9E9]];
	VAR robtarget OpenholeUD_1651 := [[389.37, -6.3, 188.73], [-0.218262, 0.672578, 0.691627, 0.147147], [0,0,0,0], [9E9, 9E9, 9E9, 9E9, 9E9, 9E9]];
	VAR robtarget OpenholeUD_1652 := [[393.34, -6.3, 188.24], [-0.208983, 0.675519, 0.693807, 0.136496], [0,0,0,0], [9E9, 9E9, 9E9, 9E9, 9E9, 9E9]];
	VAR robtarget OpenholeUD_1653 := [[397.31, -6.3, 187.76], [-0.199328, 0.678431, 0.695881, 0.125499], [0,0,0,0], [9E9, 9E9, 9E9, 9E9, 9E9, 9E9]];
	VAR robtarget OpenholeUD_1654 := [[401.28, -6.3, 187.27], [-0.189296, 0.681298, 0.69783, 0.114163], [0,0,0,0], [9E9, 9E9, 9E9, 9E9, 9E9, 9E9]];
	VAR robtarget OpenholeUD_1655 := [[405.25, -6.3, 186.78], [-0.178887, 0.684105, 0.699638, 0.102499], [0,0,0,0], [9E9, 9E9, 9E9, 9E9, 9E9, 9E9]];
	VAR robtarget OpenholeUD_1656 := [[409.22, -6.3, 186.3], [-0.168104, 0.686834, 0.701289, 0.090521], [0,0,0,0], [9E9, 9E9, 9E9, 9E9, 9E9, 9E9]];
	VAR robtarget OpenholeUD_1657 := [[413.19, -6.3, 185.81], [-0.156955, 0.689467, 0.702764, 0.078248], [0,0,0,0], [9E9, 9E9, 9E9, 9E9, 9E9, 9E9]];
	VAR robtarget OpenholeUD_1658 := [[417.16, -6.3, 185.33], [-0.14545, 0.691986, 0.704048, 0.065701], [0,0,0,0], [9E9, 9E9, 9E9, 9E9, 9E9, 9E9]];
	VAR robtarget OpenholeUD_1659 := [[421.13, -6.3, 184.84], [-0.133605, 0.69437, 0.705125, 0.052907], [0,0,0,0], [9E9, 9E9, 9E9, 9E9, 9E9, 9E9]];
	VAR robtarget OpenholeUD_1660 := [[425.1, -6.3, 184.35], [-0.121439, 0.696601, 0.70598, 0.039895], [0,0,0,0], [9E9, 9E9, 9E9, 9E9, 9E9, 9E9]];
	VAR robtarget OpenholeUD_1661 := [[429.07, -6.3, 183.87], [-0.108975, 0.698659, 0.706603, 0.0267], [0,0,0,0], [9E9, 9E9, 9E9, 9E9, 9E9, 9E9]];
	VAR robtarget OpenholeUD_1662 := [[433.04, -6.3, 183.38], [-0.096242, 0.700527, 0.706981, 0.013359], [0,0,0,0], [9E9, 9E9, 9E9, 9E9, 9E9, 9E9]];
	VAR robtarget OpenholeUD_1663 := [[437.01, -6.3, 182.89], [-0.083271, 0.702187, 0.707107, -0.000089], [0,0,0,0], [9E9, 9E9, 9E9, 9E9, 9E9, 9E9]];
	VAR robtarget OpenholeUD_1664 := [[440.98, -6.3, 182.41], [-0.070099, 0.703624, 0.706976, -0.0136], [0,0,0,0], [9E9, 9E9, 9E9, 9E9, 9E9, 9E9]];
	VAR robtarget OpenholeUD_1665 := [[444.95, -6.3, 181.92], [-0.056764, 0.704825, 0.706586, -0.027133], [0,0,0,0], [9E9, 9E9, 9E9, 9E9, 9E9, 9E9]];
	VAR robtarget OpenholeUD_1666 := [[448.92, -6.3, 181.43], [-0.043308, 0.705779, 0.705938, -0.040641], [0,0,0,0], [9E9, 9E9, 9E9, 9E9, 9E9, 9E9]];
	VAR robtarget OpenholeUD_1667 := [[452.89, -6.3, 180.95], [-0.029775, 0.70648, 0.705036, -0.054081], [0,0,0,0], [9E9, 9E9, 9E9, 9E9, 9E9, 9E9]];
	VAR robtarget OpenholeUD_1668 := [[456.86, -6.3, 180.46], [-0.016209, 0.706921, 0.703886, -0.06741], [0,0,0,0], [9E9, 9E9, 9E9, 9E9, 9E9, 9E9]];
	VAR robtarget OpenholeUD_1669 := [[460.83, -6.3, 179.97], [-0.002656, 0.707102, 0.7025, -0.080585], [0,0,0,0], [9E9, 9E9, 9E9, 9E9, 9E9, 9E9]];
	VAR robtarget OpenholeUD_1670 := [[464.8, -6.3, 179.49], [0.010841, 0.707024, 0.700889, -0.093568], [0,0,0,0], [9E9, 9E9, 9E9, 9E9, 9E9, 9E9]];
	VAR robtarget OpenholeUD_1671 := [[468.78, -6.3, 179], [0.024238, 0.706691, 0.699068, -0.106322], [0,0,0,0], [9E9, 9E9, 9E9, 9E9, 9E9, 9E9]];
	VAR robtarget OpenholeUD_1672 := [[472.75, -6.3, 178.51], [0.037495, 0.706112, 0.697053, -0.118815], [0,0,0,0], [9E9, 9E9, 9E9, 9E9, 9E9, 9E9]];
	VAR robtarget OpenholeUD_1673 := [[476.72, -6.3, 178.03], [0.050574, 0.705296, 0.694863, -0.131018], [0,0,0,0], [9E9, 9E9, 9E9, 9E9, 9E9, 9E9]];
	VAR robtarget OpenholeUD_1674 := [[480.69, -6.3, 177.54], [0.063439, 0.704255, 0.692515, -0.142907], [0,0,0,0], [9E9, 9E9, 9E9, 9E9, 9E9, 9E9]];
	VAR robtarget OpenholeUD_1675 := [[484.66, -6.3, 177.05], [0.07606, 0.703004, 0.69003, -0.154462], [0,0,0,0], [9E9, 9E9, 9E9, 9E9, 9E9, 9E9]];
	VAR robtarget OpenholeUD_1676 := [[488.63, -6.3, 176.57], [0.08841, 0.701558, 0.687426, -0.165666], [0,0,0,0], [9E9, 9E9, 9E9, 9E9, 9E9, 9E9]];
	VAR robtarget OpenholeUD_1677 := [[492.6, -6.3, 176.08], [0.100465, 0.699933, 0.684722, -0.176508], [0,0,0,0], [9E9, 9E9, 9E9, 9E9, 9E9, 9E9]];
	VAR robtarget OpenholeUD_1678 := [[496.57, -6.3, 175.6], [0.112207, 0.698147, 0.681937, -0.186981], [0,0,0,0], [9E9, 9E9, 9E9, 9E9, 9E9, 9E9]];
	VAR robtarget OpenholeUD_1679 := [[500.54, -6.3, 175.11], [0.123621, 0.696217, 0.679088, -0.197079], [0,0,0,0], [9E9, 9E9, 9E9, 9E9, 9E9, 9E9]];
	VAR robtarget OpenholeUD_1680 := [[504.51, -6.3, 174.62], [0.134696, 0.694159, 0.67619, -0.206801], [0,0,0,0], [9E9, 9E9, 9E9, 9E9, 9E9, 9E9]];
	VAR robtarget OpenholeUD_1681 := [[509.32, -6.3, 174.03], [0.183051, 0.683002, 0.683002, -0.183051], [0,0,0,0], [9E9, 9E9, 9E9, 9E9, 9E9, 9E9]];
	VAR robtarget OpenholeUD_1682 := [[513.32, -6.3, 174.02], [0.183051, 0.683002, 0.683002, -0.183051], [0,0,0,0], [9E9, 9E9, 9E9, 9E9, 9E9, 9E9]];
	VAR robtarget OpenholeUD_1683 := [[517.32, -6.3, 174.01], [0.183051, 0.683002, 0.683002, -0.183051], [0,0,0,0], [9E9, 9E9, 9E9, 9E9, 9E9, 9E9]];
	VAR robtarget OpenholeUD_1684 := [[521.32, -6.3, 173.99], [0.183051, 0.683002, 0.683002, -0.183051], [0,0,0,0], [9E9, 9E9, 9E9, 9E9, 9E9, 9E9]];
	VAR robtarget OpenholeUD_1685 := [[525.32, -6.3, 173.98], [0.183051, 0.683002, 0.683002, -0.183051], [0,0,0,0], [9E9, 9E9, 9E9, 9E9, 9E9, 9E9]];
	VAR robtarget OpenholeUD_1686 := [[529.32, -6.3, 173.97], [0.183051, 0.683002, 0.683002, -0.183051], [0,0,0,0], [9E9, 9E9, 9E9, 9E9, 9E9, 9E9]];
	VAR robtarget OpenholeUD_1687 := [[529.32, -6.3, 173.97], [0.183051, 0.683002, 0.683002, -0.183051], [0,0,0,0], [9E9, 9E9, 9E9, 9E9, 9E9, 9E9]];
	VAR robtarget OpenholeUD_1688 := [[529.33, -7.5, 174.66], [0.183051, 0.683002, 0.683002, -0.183051], [0,0,0,0], [9E9, 9E9, 9E9, 9E9, 9E9, 9E9]];
	VAR robtarget OpenholeUD_1689 := [[525.33, -7.5, 174.67], [0.183051, 0.683002, 0.683002, -0.183051], [0,0,0,0], [9E9, 9E9, 9E9, 9E9, 9E9, 9E9]];
	VAR robtarget OpenholeUD_1690 := [[521.33, -7.5, 174.69], [0.183051, 0.683002, 0.683002, -0.183051], [0,0,0,0], [9E9, 9E9, 9E9, 9E9, 9E9, 9E9]];
	VAR robtarget OpenholeUD_1691 := [[517.33, -7.5, 174.7], [0.183051, 0.683002, 0.683002, -0.183051], [0,0,0,0], [9E9, 9E9, 9E9, 9E9, 9E9, 9E9]];
	VAR robtarget OpenholeUD_1692 := [[513.33, -7.5, 174.71], [0.183051, 0.683002, 0.683002, -0.183051], [0,0,0,0], [9E9, 9E9, 9E9, 9E9, 9E9, 9E9]];
	VAR robtarget OpenholeUD_1693 := [[509.33, -7.5, 174.72], [0.183051, 0.683002, 0.683002, -0.183051], [0,0,0,0], [9E9, 9E9, 9E9, 9E9, 9E9, 9E9]];
	VAR robtarget OpenholeUD_1694 := [[505.35, -7.5, 175.17], [0.140489, 0.69301, 0.676613, -0.205413], [0,0,0,0], [9E9, 9E9, 9E9, 9E9, 9E9, 9E9]];
	VAR robtarget OpenholeUD_1695 := [[501.37, -7.5, 175.61], [0.129537, 0.69514, 0.679489, -0.195689], [0,0,0,0], [9E9, 9E9, 9E9, 9E9, 9E9, 9E9]];
	VAR robtarget OpenholeUD_1696 := [[497.4, -7.5, 176.05], [0.118242, 0.697151, 0.682317, -0.185591], [0,0,0,0], [9E9, 9E9, 9E9, 9E9, 9E9, 9E9]];
	VAR robtarget OpenholeUD_1697 := [[493.42, -7.5, 176.49], [0.106612, 0.699024, 0.685079, -0.175119], [0,0,0,0], [9E9, 9E9, 9E9, 9E9, 9E9, 9E9]];
	VAR robtarget OpenholeUD_1698 := [[489.45, -7.5, 176.93], [0.094662, 0.700742, 0.687759, -0.164277], [0,0,0,0], [9E9, 9E9, 9E9, 9E9, 9E9, 9E9]];
	VAR robtarget OpenholeUD_1699 := [[485.47, -7.5, 177.37], [0.082409, 0.702288, 0.690339, -0.153074], [0,0,0,0], [9E9, 9E9, 9E9, 9E9, 9E9, 9E9]];
	VAR robtarget OpenholeUD_1700 := [[481.5, -7.5, 177.81], [0.069874, 0.703646, 0.6928, -0.14152], [0,0,0,0], [9E9, 9E9, 9E9, 9E9, 9E9, 9E9]];
	VAR robtarget OpenholeUD_1701 := [[477.52, -7.5, 178.25], [0.057085, 0.704799, 0.695123, -0.129631], [0,0,0,0], [9E9, 9E9, 9E9, 9E9, 9E9, 9E9]];
	VAR robtarget OpenholeUD_1702 := [[473.55, -7.5, 178.7], [0.044069, 0.705732, 0.697288, -0.117428], [0,0,0,0], [9E9, 9E9, 9E9, 9E9, 9E9, 9E9]];
	VAR robtarget OpenholeUD_1703 := [[469.57, -7.5, 179.14], [0.030862, 0.706433, 0.699277, -0.104934], [0,0,0,0], [9E9, 9E9, 9E9, 9E9, 9E9, 9E9]];
	VAR robtarget OpenholeUD_1704 := [[465.59, -7.5, 179.58], [0.0175, 0.70689, 0.701073, -0.092178], [0,0,0,0], [9E9, 9E9, 9E9, 9E9, 9E9, 9E9]];
	VAR robtarget OpenholeUD_1705 := [[461.62, -7.5, 180.02], [0.004024, 0.707095, 0.702658, -0.079191], [0,0,0,0], [9E9, 9E9, 9E9, 9E9, 9E9, 9E9]];
	VAR robtarget OpenholeUD_1706 := [[457.64, -7.5, 180.46], [-0.009526, 0.707043, 0.704019, -0.066012], [0,0,0,0], [9E9, 9E9, 9E9, 9E9, 9E9, 9E9]];
	VAR robtarget OpenholeUD_1707 := [[453.67, -7.5, 180.9], [-0.023103, 0.706729, 0.705142, -0.052677], [0,0,0,0], [9E9, 9E9, 9E9, 9E9, 9E9, 9E9]];
	VAR robtarget OpenholeUD_1708 := [[449.69, -7.5, 181.34], [-0.036664, 0.706156, 0.706018, -0.039229], [0,0,0,0], [9E9, 9E9, 9E9, 9E9, 9E9, 9E9]];
	VAR robtarget OpenholeUD_1709 := [[445.72, -7.5, 181.78], [-0.050162, 0.705325, 0.706639, -0.025711], [0,0,0,0], [9E9, 9E9, 9E9, 9E9, 9E9, 9E9]];
	VAR robtarget OpenholeUD_1710 := [[441.74, -7.5, 182.23], [-0.063556, 0.704245, 0.707002, -0.012168], [0,0,0,0], [9E9, 9E9, 9E9, 9E9, 9E9, 9E9]];
	VAR robtarget OpenholeUD_1711 := [[437.77, -7.5, 182.67], [-0.076801, 0.702924, 0.707105, 0.001355], [0,0,0,0], [9E9, 9E9, 9E9, 9E9, 9E9, 9E9]];
	VAR robtarget OpenholeUD_1712 := [[433.79, -7.5, 183.11], [-0.089857, 0.701374, 0.706952, 0.014816], [0,0,0,0], [9E9, 9E9, 9E9, 9E9, 9E9, 9E9]];
	VAR robtarget OpenholeUD_1713 := [[429.81, -7.5, 183.55], [-0.102689, 0.699611, 0.706545, 0.028171], [0,0,0,0], [9E9, 9E9, 9E9, 9E9, 9E9, 9E9]];
	VAR robtarget OpenholeUD_1714 := [[425.84, -7.5, 183.99], [-0.115261, 0.697649, 0.705895, 0.041381], [0,0,0,0], [9E9, 9E9, 9E9, 9E9, 9E9, 9E9]];
	VAR robtarget OpenholeUD_1715 := [[421.86, -7.5, 184.43], [-0.127546, 0.695508, 0.70501, 0.054408], [0,0,0,0], [9E9, 9E9, 9E9, 9E9, 9E9, 9E9]];
	VAR robtarget OpenholeUD_1716 := [[417.89, -7.5, 184.87], [-0.139518, 0.693206, 0.703905, 0.067217], [0,0,0,0], [9E9, 9E9, 9E9, 9E9, 9E9, 9E9]];
	VAR robtarget OpenholeUD_1717 := [[413.91, -7.5, 185.31], [-0.151156, 0.690762, 0.702592, 0.07978], [0,0,0,0], [9E9, 9E9, 9E9, 9E9, 9E9, 9E9]];
	VAR robtarget OpenholeUD_1718 := [[409.94, -7.5, 185.76], [-0.162443, 0.688195, 0.701087, 0.092068], [0,0,0,0], [9E9, 9E9, 9E9, 9E9, 9E9, 9E9]];
	VAR robtarget OpenholeUD_1719 := [[405.96, -7.5, 186.2], [-0.173368, 0.685524, 0.699408, 0.10406], [0,0,0,0], [9E9, 9E9, 9E9, 9E9, 9E9, 9E9]];
	VAR robtarget OpenholeUD_1720 := [[401.98, -7.5, 186.64], [-0.183922, 0.682769, 0.697571, 0.115737], [0,0,0,0], [9E9, 9E9, 9E9, 9E9, 9E9, 9E9]];
	VAR robtarget OpenholeUD_1721 := [[398.01, -7.5, 187.08], [-0.1941, 0.679945, 0.695593, 0.127085], [0,0,0,0], [9E9, 9E9, 9E9, 9E9, 9E9, 9E9]];
	VAR robtarget OpenholeUD_1722 := [[394.03, -7.5, 187.52], [-0.203901, 0.67707, 0.693492, 0.138092], [0,0,0,0], [9E9, 9E9, 9E9, 9E9, 9E9, 9E9]];
	VAR robtarget OpenholeUD_1723 := [[389.37, -7.5, 188.04], [-0.214926, 0.673652, 0.69089, 0.15057], [0,0,0,0], [9E9, 9E9, 9E9, 9E9, 9E9, 9E9]];
	VAR robtarget OpenholeUD_1724 := [[385.37, -7.5, 188.05], [-0.183051, 0.683002, 0.683002, 0.183051], [0,0,0,0], [9E9, 9E9, 9E9, 9E9, 9E9, 9E9]];
	VAR robtarget OpenholeUD_1725 := [[381.37, -7.5, 188.06], [-0.183051, 0.683002, 0.683002, 0.183051], [0,0,0,0], [9E9, 9E9, 9E9, 9E9, 9E9, 9E9]];
	VAR robtarget OpenholeUD_1726 := [[377.37, -7.5, 188.08], [-0.183051, 0.683002, 0.683002, 0.183051], [0,0,0,0], [9E9, 9E9, 9E9, 9E9, 9E9, 9E9]];
	VAR robtarget OpenholeUD_1727 := [[373.37, -7.5, 188.09], [-0.183051, 0.683002, 0.683002, 0.183051], [0,0,0,0], [9E9, 9E9, 9E9, 9E9, 9E9, 9E9]];
	VAR robtarget OpenholeUD_1728 := [[369.37, -7.5, 188.1], [-0.183051, 0.683002, 0.683002, 0.183051], [0,0,0,0], [9E9, 9E9, 9E9, 9E9, 9E9, 9E9]];
	VAR robtarget OpenholeUD_1729 := [[369.37, -7.5, 188.1], [-0.183051, 0.683002, 0.683002, 0.183051], [0,0,0,0], [9E9, 9E9, 9E9, 9E9, 9E9, 9E9]];
	VAR robtarget OpenholeUD_1730 := [[369.36, -8.7, 187.41], [-0.183051, 0.683002, 0.683002, 0.183051], [0,0,0,0], [9E9, 9E9, 9E9, 9E9, 9E9, 9E9]];
	VAR robtarget OpenholeUD_1731 := [[373.36, -8.7, 187.4], [-0.183051, 0.683002, 0.683002, 0.183051], [0,0,0,0], [9E9, 9E9, 9E9, 9E9, 9E9, 9E9]];
	VAR robtarget OpenholeUD_1732 := [[377.36, -8.7, 187.38], [-0.183051, 0.683002, 0.683002, 0.183051], [0,0,0,0], [9E9, 9E9, 9E9, 9E9, 9E9, 9E9]];
	VAR robtarget OpenholeUD_1733 := [[381.36, -8.7, 187.37], [-0.183051, 0.683002, 0.683002, 0.183051], [0,0,0,0], [9E9, 9E9, 9E9, 9E9, 9E9, 9E9]];
	VAR robtarget OpenholeUD_1734 := [[385.36, -8.7, 187.36], [-0.183051, 0.683002, 0.683002, 0.183051], [0,0,0,0], [9E9, 9E9, 9E9, 9E9, 9E9, 9E9]];
	VAR robtarget OpenholeUD_1735 := [[389.36, -8.7, 187.34], [-0.211579, 0.674711, 0.690134, 0.153995], [0,0,0,0], [9E9, 9E9, 9E9, 9E9, 9E9, 9E9]];
	VAR robtarget OpenholeUD_1736 := [[393.35, -8.7, 186.95], [-0.202138, 0.677599, 0.692403, 0.143449], [0,0,0,0], [9E9, 9E9, 9E9, 9E9, 9E9, 9E9]];
	VAR robtarget OpenholeUD_1737 := [[397.33, -8.7, 186.55], [-0.192323, 0.68045, 0.694572, 0.132553], [0,0,0,0], [9E9, 9E9, 9E9, 9E9, 9E9, 9E9]];
	VAR robtarget OpenholeUD_1738 := [[401.31, -8.7, 186.16], [-0.182131, 0.683248, 0.696623, 0.121312], [0,0,0,0], [9E9, 9E9, 9E9, 9E9, 9E9, 9E9]];
	VAR robtarget OpenholeUD_1739 := [[405.29, -8.7, 185.76], [-0.171563, 0.685978, 0.69854, 0.109737], [0,0,0,0], [9E9, 9E9, 9E9, 9E9, 9E9, 9E9]];
	VAR robtarget OpenholeUD_1740 := [[409.27, -8.7, 185.37], [-0.160626, 0.688621, 0.700305, 0.097841], [0,0,0,0], [9E9, 9E9, 9E9, 9E9, 9E9, 9E9]];
	VAR robtarget OpenholeUD_1741 := [[413.25, -8.7, 184.97], [-0.149326, 0.69116, 0.701902, 0.08564], [0,0,0,0], [9E9, 9E9, 9E9, 9E9, 9E9, 9E9]];
	VAR robtarget OpenholeUD_1742 := [[417.23, -8.7, 184.57], [-0.137677, 0.693574, 0.703312, 0.073157], [0,0,0,0], [9E9, 9E9, 9E9, 9E9, 9E9, 9E9]];
	VAR robtarget OpenholeUD_1743 := [[421.21, -8.7, 184.18], [-0.125693, 0.695846, 0.704521, 0.060416], [0,0,0,0], [9E9, 9E9, 9E9, 9E9, 9E9, 9E9]];
	VAR robtarget OpenholeUD_1744 := [[425.19, -8.7, 183.78], [-0.113398, 0.697955, 0.705513, 0.047448], [0,0,0,0], [9E9, 9E9, 9E9, 9E9, 9E9, 9E9]];
	VAR robtarget OpenholeUD_1745 := [[429.17, -8.7, 183.39], [-0.100814, 0.699883, 0.706275, 0.034284], [0,0,0,0], [9E9, 9E9, 9E9, 9E9, 9E9, 9E9]];
	VAR robtarget OpenholeUD_1746 := [[433.15, -8.7, 182.99], [-0.087972, 0.701613, 0.706796, 0.020962], [0,0,0,0], [9E9, 9E9, 9E9, 9E9, 9E9, 9E9]];
	VAR robtarget OpenholeUD_1747 := [[437.13, -8.7, 182.6], [-0.074905, 0.703128, 0.707067, 0.007521], [0,0,0,0], [9E9, 9E9, 9E9, 9E9, 9E9, 9E9]];
	VAR robtarget OpenholeUD_1748 := [[441.11, -8.7, 182.2], [-0.06165, 0.704414, 0.707081, -0.005997], [0,0,0,0], [9E9, 9E9, 9E9, 9E9, 9E9, 9E9]];
	VAR robtarget OpenholeUD_1749 := [[445.09, -8.7, 181.8], [-0.048246, 0.705459, 0.706837, -0.019548], [0,0,0,0], [9E9, 9E9, 9E9, 9E9, 9E9, 9E9]];
	VAR robtarget OpenholeUD_1750 := [[449.07, -8.7, 181.41], [-0.034737, 0.706253, 0.706332, -0.033089], [0,0,0,0], [9E9, 9E9, 9E9, 9E9, 9E9, 9E9]];
	VAR robtarget OpenholeUD_1751 := [[453.05, -8.7, 181.01], [-0.021167, 0.70679, 0.705571, -0.046573], [0,0,0,0], [9E9, 9E9, 9E9, 9E9, 9E9, 9E9]];
	VAR robtarget OpenholeUD_1752 := [[457.03, -8.7, 180.62], [-0.00758, 0.707066, 0.70456, -0.059958], [0,0,0,0], [9E9, 9E9, 9E9, 9E9, 9E9, 9E9]];
	VAR robtarget OpenholeUD_1753 := [[461.01, -8.7, 180.22], [0.005979, 0.707082, 0.703308, -0.073201], [0,0,0,0], [9E9, 9E9, 9E9, 9E9, 9E9, 9E9]];
	VAR robtarget OpenholeUD_1754 := [[464.99, -8.7, 179.83], [0.019464, 0.706839, 0.701825, -0.086262], [0,0,0,0], [9E9, 9E9, 9E9, 9E9, 9E9, 9E9]];
	VAR robtarget OpenholeUD_1755 := [[468.97, -8.7, 179.43], [0.032834, 0.706344, 0.700127, -0.099104], [0,0,0,0], [9E9, 9E9, 9E9, 9E9, 9E9, 9E9]];
	VAR robtarget OpenholeUD_1756 := [[472.95, -8.7, 179.03], [0.046049, 0.705606, 0.69823, -0.111694], [0,0,0,0], [9E9, 9E9, 9E9, 9E9, 9E9, 9E9]];
	VAR robtarget OpenholeUD_1757 := [[476.93, -8.7, 178.64], [0.059071, 0.704635, 0.696149, -0.124002], [0,0,0,0], [9E9, 9E9, 9E9, 9E9, 9E9, 9E9]];
	VAR robtarget OpenholeUD_1758 := [[480.91, -8.7, 178.24], [0.071866, 0.703445, 0.693904, -0.136002], [0,0,0,0], [9E9, 9E9, 9E9, 9E9, 9E9, 9E9]];
	VAR robtarget OpenholeUD_1759 := [[484.89, -8.7, 177.85], [0.084404, 0.702051, 0.691514, -0.147674], [0,0,0,0], [9E9, 9E9, 9E9, 9E9, 9E9, 9E9]];
	VAR robtarget OpenholeUD_1760 := [[488.87, -8.7, 177.45], [0.09666, 0.700469, 0.688998, -0.159001], [0,0,0,0], [9E9, 9E9, 9E9, 9E9, 9E9, 9E9]];
	VAR robtarget OpenholeUD_1761 := [[492.85, -8.7, 177.06], [0.108611, 0.698716, 0.686375, -0.16997], [0,0,0,0], [9E9, 9E9, 9E9, 9E9, 9E9, 9E9]];
	VAR robtarget OpenholeUD_1762 := [[496.84, -8.7, 176.66], [0.120241, 0.696809, 0.683662, -0.180571], [0,0,0,0], [9E9, 9E9, 9E9, 9E9, 9E9, 9E9]];
	VAR robtarget OpenholeUD_1763 := [[500.82, -8.7, 176.26], [0.131535, 0.694765, 0.680878, -0.1908], [0,0,0,0], [9E9, 9E9, 9E9, 9E9, 9E9, 9E9]];
	VAR robtarget OpenholeUD_1764 := [[504.8, -8.7, 175.87], [0.142483, 0.692603, 0.678039, -0.200655], [0,0,0,0], [9E9, 9E9, 9E9, 9E9, 9E9, 9E9]];
	VAR robtarget OpenholeUD_1765 := [[509.33, -8.7, 175.42], [0.183051, 0.683002, 0.683002, -0.183051], [0,0,0,0], [9E9, 9E9, 9E9, 9E9, 9E9, 9E9]];
	VAR robtarget OpenholeUD_1766 := [[513.33, -8.7, 175.41], [0.183051, 0.683002, 0.683002, -0.183051], [0,0,0,0], [9E9, 9E9, 9E9, 9E9, 9E9, 9E9]];
	VAR robtarget OpenholeUD_1767 := [[517.33, -8.7, 175.39], [0.183051, 0.683002, 0.683002, -0.183051], [0,0,0,0], [9E9, 9E9, 9E9, 9E9, 9E9, 9E9]];
	VAR robtarget OpenholeUD_1768 := [[521.33, -8.7, 175.38], [0.183051, 0.683002, 0.683002, -0.183051], [0,0,0,0], [9E9, 9E9, 9E9, 9E9, 9E9, 9E9]];
	VAR robtarget OpenholeUD_1769 := [[529.33, -8.7, 175.36], [0.183051, 0.683002, 0.683002, -0.183051], [0,0,0,0], [9E9, 9E9, 9E9, 9E9, 9E9, 9E9]];
	VAR robtarget OpenholeUD_1770 := [[529.33, -8.7, 175.36], [0.183051, 0.683002, 0.683002, -0.183051], [0,0,0,0], [9E9, 9E9, 9E9, 9E9, 9E9, 9E9]];
	VAR robtarget OpenholeUD_1771 := [[529.33, -9.9, 176.05], [0.183051, 0.683002, 0.683002, -0.183051], [0,0,0,0], [9E9, 9E9, 9E9, 9E9, 9E9, 9E9]];
	VAR robtarget OpenholeUD_1772 := [[525.33, -9.9, 176.06], [0.183051, 0.683002, 0.683002, -0.183051], [0,0,0,0], [9E9, 9E9, 9E9, 9E9, 9E9, 9E9]];
	VAR robtarget OpenholeUD_1773 := [[521.33, -9.9, 176.07], [0.183051, 0.683002, 0.683002, -0.183051], [0,0,0,0], [9E9, 9E9, 9E9, 9E9, 9E9, 9E9]];
	VAR robtarget OpenholeUD_1774 := [[517.33, -9.9, 176.09], [0.183051, 0.683002, 0.683002, -0.183051], [0,0,0,0], [9E9, 9E9, 9E9, 9E9, 9E9, 9E9]];
	VAR robtarget OpenholeUD_1775 := [[509.33, -9.9, 176.11], [0.183051, 0.683002, 0.683002, -0.183051], [0,0,0,0], [9E9, 9E9, 9E9, 9E9, 9E9, 9E9]];
	VAR robtarget OpenholeUD_1776 := [[505.35, -9.9, 176.46], [0.14746, 0.69156, 0.678656, -0.198561], [0,0,0,0], [9E9, 9E9, 9E9, 9E9, 9E9, 9E9]];
	VAR robtarget OpenholeUD_1777 := [[501.36, -9.9, 176.81], [0.136615, 0.693784, 0.681469, -0.188679], [0,0,0,0], [9E9, 9E9, 9E9, 9E9, 9E9, 9E9]];
	VAR robtarget OpenholeUD_1778 := [[497.38, -9.9, 177.16], [0.12542, 0.695895, 0.684226, -0.178424], [0,0,0,0], [9E9, 9E9, 9E9, 9E9, 9E9, 9E9]];
	VAR robtarget OpenholeUD_1779 := [[493.39, -9.9, 177.51], [0.113885, 0.697876, 0.686909, -0.167797], [0,0,0,0], [9E9, 9E9, 9E9, 9E9, 9E9, 9E9]];
	VAR robtarget OpenholeUD_1780 := [[489.41, -9.9, 177.86], [0.102022, 0.699708, 0.689502, -0.156804], [0,0,0,0], [9E9, 9E9, 9E9, 9E9, 9E9, 9E9]];
	VAR robtarget OpenholeUD_1781 := [[485.42, -9.9, 178.21], [0.089848, 0.701375, 0.691985, -0.145454], [0,0,0,0], [9E9, 9E9, 9E9, 9E9, 9E9, 9E9]];
	VAR robtarget OpenholeUD_1782 := [[481.44, -9.9, 178.56], [0.077383, 0.70286, 0.69434, -0.133759], [0,0,0,0], [9E9, 9E9, 9E9, 9E9, 9E9, 9E9]];
	VAR robtarget OpenholeUD_1783 := [[477.45, -9.9, 178.91], [0.064653, 0.704145, 0.696549, -0.121737], [0,0,0,0], [9E9, 9E9, 9E9, 9E9, 9E9, 9E9]];
	VAR robtarget OpenholeUD_1784 := [[473.47, -9.9, 179.26], [0.051686, 0.705215, 0.698591, -0.109409], [0,0,0,0], [9E9, 9E9, 9E9, 9E9, 9E9, 9E9]];
	VAR robtarget OpenholeUD_1785 := [[469.48, -9.9, 179.61], [0.038516, 0.706057, 0.70045, -0.0968], [0,0,0,0], [9E9, 9E9, 9E9, 9E9, 9E9, 9E9]];
	VAR robtarget OpenholeUD_1786 := [[465.5, -9.9, 179.96], [0.025178, 0.706658, 0.702107, -0.08394], [0,0,0,0], [9E9, 9E9, 9E9, 9E9, 9E9, 9E9]];
	VAR robtarget OpenholeUD_1787 := [[461.51, -9.9, 180.31], [0.011713, 0.70701, 0.703547, -0.070863], [0,0,0,0], [9E9, 9E9, 9E9, 9E9, 9E9, 9E9]];
	VAR robtarget OpenholeUD_1788 := [[457.53, -9.9, 180.66], [-0.001837, 0.707104, 0.704756, -0.057605], [0,0,0,0], [9E9, 9E9, 9E9, 9E9, 9E9, 9E9]];
	VAR robtarget OpenholeUD_1789 := [[453.55, -9.9, 181.01], [-0.015429, 0.706938, 0.705724, -0.044207], [0,0,0,0], [9E9, 9E9, 9E9, 9E9, 9E9, 9E9]];
	VAR robtarget OpenholeUD_1790 := [[449.56, -9.9, 181.36], [-0.029018, 0.706511, 0.70644, -0.030712], [0,0,0,0], [9E9, 9E9, 9E9, 9E9, 9E9, 9E9]];
	VAR robtarget OpenholeUD_1791 := [[445.58, -9.9, 181.71], [-0.042557, 0.705825, 0.706898, -0.017162], [0,0,0,0], [9E9, 9E9, 9E9, 9E9, 9E9, 9E9]];
	VAR robtarget OpenholeUD_1792 := [[441.59, -9.9, 182.06], [-0.056004, 0.704885, 0.707098, -0.003602], [0,0,0,0], [9E9, 9E9, 9E9, 9E9, 9E9, 9E9]];
	VAR robtarget OpenholeUD_1793 := [[437.61, -9.9, 182.41], [-0.069314, 0.703701, 0.707037, 0.009922], [0,0,0,0], [9E9, 9E9, 9E9, 9E9, 9E9, 9E9]];
	VAR robtarget OpenholeUD_1794 := [[433.62, -9.9, 182.76], [-0.082447, 0.702284, 0.706721, 0.023367], [0,0,0,0], [9E9, 9E9, 9E9, 9E9, 9E9, 9E9]];
	VAR robtarget OpenholeUD_1795 := [[429.64, -9.9, 183.11], [-0.095365, 0.700646, 0.706154, 0.036692], [0,0,0,0], [9E9, 9E9, 9E9, 9E9, 9E9, 9E9]];
	VAR robtarget OpenholeUD_1796 := [[425.65, -9.9, 183.46], [-0.108034, 0.698805, 0.705347, 0.049855], [0,0,0,0], [9E9, 9E9, 9E9, 9E9, 9E9, 9E9]];
	VAR robtarget OpenholeUD_1797 := [[421.67, -9.9, 183.81], [-0.120424, 0.696777, 0.704311, 0.062822], [0,0,0,0], [9E9, 9E9, 9E9, 9E9, 9E9, 9E9]];
	VAR robtarget OpenholeUD_1798 := [[417.68, -9.9, 184.16], [-0.132507, 0.69458, 0.703058, 0.075559], [0,0,0,0], [9E9, 9E9, 9E9, 9E9, 9E9, 9E9]];
	VAR robtarget OpenholeUD_1799 := [[413.7, -9.9, 184.51], [-0.144263, 0.692234, 0.701605, 0.088036], [0,0,0,0], [9E9, 9E9, 9E9, 9E9, 9E9, 9E9]];
	VAR robtarget OpenholeUD_1800 := [[409.71, -9.9, 184.86], [-0.155673, 0.689758, 0.699967, 0.100228], [0,0,0,0], [9E9, 9E9, 9E9, 9E9, 9E9, 9E9]];
	VAR robtarget OpenholeUD_1801 := [[405.73, -9.9, 185.21], [-0.166726, 0.68717, 0.698162, 0.112114], [0,0,0,0], [9E9, 9E9, 9E9, 9E9, 9E9, 9E9]];
	VAR robtarget OpenholeUD_1802 := [[401.74, -9.9, 185.56], [-0.17741, 0.684489, 0.696207, 0.123677], [0,0,0,0], [9E9, 9E9, 9E9, 9E9, 9E9, 9E9]];
	VAR robtarget OpenholeUD_1803 := [[397.76, -9.9, 185.91], [-0.187721, 0.681734, 0.694119, 0.134904], [0,0,0,0], [9E9, 9E9, 9E9, 9E9, 9E9, 9E9]];
	VAR robtarget OpenholeUD_1804 := [[393.78, -9.9, 186.26], [-0.197656, 0.67892, 0.691915, 0.145784], [0,0,0,0], [9E9, 9E9, 9E9, 9E9, 9E9, 9E9]];
	VAR robtarget OpenholeUD_1805 := [[389.36, -9.9, 186.65], [-0.208221, 0.675754, 0.689361, 0.157422], [0,0,0,0], [9E9, 9E9, 9E9, 9E9, 9E9, 9E9]];
	VAR robtarget OpenholeUD_1806 := [[385.36, -9.9, 186.66], [-0.183051, 0.683002, 0.683002, 0.183051], [0,0,0,0], [9E9, 9E9, 9E9, 9E9, 9E9, 9E9]];
	VAR robtarget OpenholeUD_1807 := [[381.36, -9.9, 186.68], [-0.183051, 0.683002, 0.683002, 0.183051], [0,0,0,0], [9E9, 9E9, 9E9, 9E9, 9E9, 9E9]];
	VAR robtarget OpenholeUD_1808 := [[377.36, -9.9, 186.69], [-0.183051, 0.683002, 0.683002, 0.183051], [0,0,0,0], [9E9, 9E9, 9E9, 9E9, 9E9, 9E9]];
	VAR robtarget OpenholeUD_1809 := [[373.36, -9.9, 186.7], [-0.183051, 0.683002, 0.683002, 0.183051], [0,0,0,0], [9E9, 9E9, 9E9, 9E9, 9E9, 9E9]];
	VAR robtarget OpenholeUD_1810 := [[369.36, -9.9, 186.71], [-0.183051, 0.683002, 0.683002, 0.183051], [0,0,0,0], [9E9, 9E9, 9E9, 9E9, 9E9, 9E9]];
	VAR robtarget OpenholeUD_1811 := [[369.36, -9.9, 186.71], [-0.183051, 0.683002, 0.683002, 0.183051], [0,0,0,0], [9E9, 9E9, 9E9, 9E9, 9E9, 9E9]];
	VAR robtarget OpenholeUD_1812 := [[369.36, -11.1, 186.02], [-0.183051, 0.683002, 0.683002, 0.183051], [0,0,0,0], [9E9, 9E9, 9E9, 9E9, 9E9, 9E9]];
	VAR robtarget OpenholeUD_1813 := [[373.36, -11.1, 186.01], [-0.183051, 0.683002, 0.683002, 0.183051], [0,0,0,0], [9E9, 9E9, 9E9, 9E9, 9E9, 9E9]];
	VAR robtarget OpenholeUD_1814 := [[377.36, -11.1, 186], [-0.183051, 0.683002, 0.683002, 0.183051], [0,0,0,0], [9E9, 9E9, 9E9, 9E9, 9E9, 9E9]];
	VAR robtarget OpenholeUD_1815 := [[381.36, -11.1, 185.98], [-0.183051, 0.683002, 0.683002, 0.183051], [0,0,0,0], [9E9, 9E9, 9E9, 9E9, 9E9, 9E9]];
	VAR robtarget OpenholeUD_1816 := [[385.36, -11.1, 185.97], [-0.183051, 0.683002, 0.683002, 0.183051], [0,0,0,0], [9E9, 9E9, 9E9, 9E9, 9E9, 9E9]];
	VAR robtarget OpenholeUD_1817 := [[389.36, -11.1, 185.96], [-0.204853, 0.676783, 0.688569, 0.16085], [0,0,0,0], [9E9, 9E9, 9E9, 9E9, 9E9, 9E9]];
	VAR robtarget OpenholeUD_1818 := [[393.35, -11.1, 185.65], [-0.195254, 0.679614, 0.690923, 0.150418], [0,0,0,0], [9E9, 9E9, 9E9, 9E9, 9E9, 9E9]];
	VAR robtarget OpenholeUD_1819 := [[397.34, -11.1, 185.35], [-0.185281, 0.682401, 0.693183, 0.139631], [0,0,0,0], [9E9, 9E9, 9E9, 9E9, 9E9, 9E9]];
	VAR robtarget OpenholeUD_1820 := [[401.33, -11.1, 185.05], [-0.174933, 0.685127, 0.695334, 0.128494], [0,0,0,0], [9E9, 9E9, 9E9, 9E9, 9E9, 9E9]];
	VAR robtarget OpenholeUD_1821 := [[405.31, -11.1, 184.74], [-0.164213, 0.687775, 0.697357, 0.117017], [0,0,0,0], [9E9, 9E9, 9E9, 9E9, 9E9, 9E9]];
	VAR robtarget OpenholeUD_1822 := [[409.3, -11.1, 184.44], [-0.153126, 0.690328, 0.699236, 0.105211], [0,0,0,0], [9E9, 9E9, 9E9, 9E9, 9E9, 9E9]];
	VAR robtarget OpenholeUD_1823 := [[413.29, -11.1, 184.13], [-0.141682, 0.692767, 0.700952, 0.093093], [0,0,0,0], [9E9, 9E9, 9E9, 9E9, 9E9, 9E9]];
	VAR robtarget OpenholeUD_1824 := [[417.28, -11.1, 183.83], [-0.129894, 0.695074, 0.702489, 0.080684], [0,0,0,0], [9E9, 9E9, 9E9, 9E9, 9E9, 9E9]];
	VAR robtarget OpenholeUD_1825 := [[421.27, -11.1, 183.52], [-0.117781, 0.697229, 0.703829, 0.068007], [0,0,0,0], [9E9, 9E9, 9E9, 9E9, 9E9, 9E9]];
	VAR robtarget OpenholeUD_1826 := [[425.26, -11.1, 183.22], [-0.105363, 0.699213, 0.704957, 0.055091], [0,0,0,0], [9E9, 9E9, 9E9, 9E9, 9E9, 9E9]];
	VAR robtarget OpenholeUD_1827 := [[429.24, -11.1, 182.92], [-0.092669, 0.701008, 0.70586, 0.041968], [0,0,0,0], [9E9, 9E9, 9E9, 9E9, 9E9, 9E9]];
	VAR robtarget OpenholeUD_1828 := [[433.23, -11.1, 182.61], [-0.079727, 0.702598, 0.706525, 0.028675], [0,0,0,0], [9E9, 9E9, 9E9, 9E9, 9E9, 9E9]];
	VAR robtarget OpenholeUD_1829 := [[437.22, -11.1, 182.31], [-0.066573, 0.703966, 0.706942, 0.01525], [0,0,0,0], [9E9, 9E9, 9E9, 9E9, 9E9, 9E9]];
	VAR robtarget OpenholeUD_1830 := [[441.21, -11.1, 182], [-0.053244, 0.705099, 0.707105, 0.001734], [0,0,0,0], [9E9, 9E9, 9E9, 9E9, 9E9, 9E9]];
	VAR robtarget OpenholeUD_1831 := [[445.2, -11.1, 181.7], [-0.039783, 0.705987, 0.707008, -0.011828], [0,0,0,0], [9E9, 9E9, 9E9, 9E9, 9E9, 9E9]];
	VAR robtarget OpenholeUD_1832 := [[449.19, -11.1, 181.39], [-0.02623, 0.70662, 0.706651, -0.025392], [0,0,0,0], [9E9, 9E9, 9E9, 9E9, 9E9, 9E9]];
	VAR robtarget OpenholeUD_1833 := [[453.17, -11.1, 181.09], [-0.012633, 0.706994, 0.706035, -0.038914], [0,0,0,0], [9E9, 9E9, 9E9, 9E9, 9E9, 9E9]];
	VAR robtarget OpenholeUD_1834 := [[457.16, -11.1, 180.78], [0.000965, 0.707106, 0.705166, -0.052348], [0,0,0,0], [9E9, 9E9, 9E9, 9E9, 9E9, 9E9]];
	VAR robtarget OpenholeUD_1835 := [[461.15, -11.1, 180.48], [0.014519, 0.706958, 0.704052, -0.065653], [0,0,0,0], [9E9, 9E9, 9E9, 9E9, 9E9, 9E9]];
	VAR robtarget OpenholeUD_1836 := [[465.14, -11.1, 180.18], [0.027983, 0.706553, 0.702704, -0.078788], [0,0,0,0], [9E9, 9E9, 9E9, 9E9, 9E9, 9E9]];
	VAR robtarget OpenholeUD_1837 := [[469.13, -11.1, 179.87], [0.041317, 0.705899, 0.701134, -0.091715], [0,0,0,0], [9E9, 9E9, 9E9, 9E9, 9E9, 9E9]];
	VAR robtarget OpenholeUD_1838 := [[473.12, -11.1, 179.57], [0.054481, 0.705005, 0.699358, -0.104399], [0,0,0,0], [9E9, 9E9, 9E9, 9E9, 9E9, 9E9]];
	VAR robtarget OpenholeUD_1839 := [[477.11, -11.1, 179.26], [0.067437, 0.703884, 0.697392, -0.116809], [0,0,0,0], [9E9, 9E9, 9E9, 9E9, 9E9, 9E9]];
	VAR robtarget OpenholeUD_1840 := [[481.09, -11.1, 178.96], [0.080154, 0.702549, 0.695255, -0.12892], [0,0,0,0], [9E9, 9E9, 9E9, 9E9, 9E9, 9E9]];
	VAR robtarget OpenholeUD_1841 := [[485.08, -11.1, 178.65], [0.092603, 0.701017, 0.692965, -0.140709], [0,0,0,0], [9E9, 9E9, 9E9, 9E9, 9E9, 9E9]];
	VAR robtarget OpenholeUD_1842 := [[489.07, -11.1, 178.35], [0.104759, 0.699304, 0.690542, -0.152159], [0,0,0,0], [9E9, 9E9, 9E9, 9E9, 9E9, 9E9]];
	VAR robtarget OpenholeUD_1843 := [[493.06, -11.1, 178.05], [0.116601, 0.697427, 0.688003, -0.163254], [0,0,0,0], [9E9, 9E9, 9E9, 9E9, 9E9, 9E9]];
	VAR robtarget OpenholeUD_1844 := [[497.05, -11.1, 177.74], [0.128113, 0.695404, 0.685368, -0.173986], [0,0,0,0], [9E9, 9E9, 9E9, 9E9, 9E9, 9E9]];
	VAR robtarget OpenholeUD_1845 := [[501.04, -11.1, 177.44], [0.139282, 0.693254, 0.682654, -0.184348], [0,0,0,0], [9E9, 9E9, 9E9, 9E9, 9E9, 9E9]];
	VAR robtarget OpenholeUD_1846 := [[505.02, -11.1, 177.13], [0.150099, 0.690992, 0.679877, -0.194337], [0,0,0,0], [9E9, 9E9, 9E9, 9E9, 9E9, 9E9]];
	VAR robtarget OpenholeUD_1847 := [[509.33, -11.1, 176.8], [0.183051, 0.683002, 0.683002, -0.183051], [0,0,0,0], [9E9, 9E9, 9E9, 9E9, 9E9, 9E9]];
	VAR robtarget OpenholeUD_1848 := [[513.33, -11.1, 176.79], [0.183051, 0.683002, 0.683002, -0.183051], [0,0,0,0], [9E9, 9E9, 9E9, 9E9, 9E9, 9E9]];
	VAR robtarget OpenholeUD_1849 := [[517.33, -11.1, 176.78], [0.183051, 0.683002, 0.683002, -0.183051], [0,0,0,0], [9E9, 9E9, 9E9, 9E9, 9E9, 9E9]];
	VAR robtarget OpenholeUD_1850 := [[521.33, -11.1, 176.77], [0.183051, 0.683002, 0.683002, -0.183051], [0,0,0,0], [9E9, 9E9, 9E9, 9E9, 9E9, 9E9]];
	VAR robtarget OpenholeUD_1851 := [[529.33, -11.1, 176.74], [0.183051, 0.683002, 0.683002, -0.183051], [0,0,0,0], [9E9, 9E9, 9E9, 9E9, 9E9, 9E9]];
	VAR robtarget OpenholeUD_1852 := [[529.34, -14.56, 178.74], [0.183051, 0.683002, 0.683002, -0.183051], [0,0,0,0], [9E9, 9E9, 9E9, 9E9, 9E9, 9E9]];
	VAR robtarget OpenholeUD_1853 := [[529.34, -18.03, 180.74], [0.183051, 0.683002, 0.683002, -0.183051], [0,0,0,0], [9E9, 9E9, 9E9, 9E9, 9E9, 9E9]];
	VAR robtarget OpenholeUD_1854 := [[529.36, -24.3, 184.36], [0.183051, 0.683002, 0.683002, -0.183051], [0,0,0,0], [9E9, 9E9, 9E9, 9E9, 9E9, 9E9]];
	VAR robtarget OpenholeUD_1855 := [[525.36, -24.3, 184.38], [0.183051, 0.683002, 0.683002, -0.183051], [0,0,0,0], [9E9, 9E9, 9E9, 9E9, 9E9, 9E9]];
	VAR robtarget OpenholeUD_1856 := [[521.36, -24.3, 184.39], [0.183051, 0.683002, 0.683002, -0.183051], [0,0,0,0], [9E9, 9E9, 9E9, 9E9, 9E9, 9E9]];
	VAR robtarget OpenholeUD_1857 := [[517.36, -24.3, 184.4], [0.183051, 0.683002, 0.683002, -0.183051], [0,0,0,0], [9E9, 9E9, 9E9, 9E9, 9E9, 9E9]];
	VAR robtarget OpenholeUD_1858 := [[513.36, -24.3, 184.41], [0.183051, 0.683002, 0.683002, -0.183051], [0,0,0,0], [9E9, 9E9, 9E9, 9E9, 9E9, 9E9]];
	VAR robtarget OpenholeUD_1859 := [[509.36, -24.3, 184.43], [0.183051, 0.683002, 0.683002, -0.183051], [0,0,0,0], [9E9, 9E9, 9E9, 9E9, 9E9, 9E9]];
	VAR robtarget OpenholeUD_1860 := [[505.36, -24.3, 184.22], [0.189301, 0.681297, 0.689475, -0.156922], [0,0,0,0], [9E9, 9E9, 9E9, 9E9, 9E9, 9E9]];
	VAR robtarget OpenholeUD_1861 := [[501.37, -24.3, 184.02], [0.179247, 0.684011, 0.691828, -0.146199], [0,0,0,0], [9E9, 9E9, 9E9, 9E9, 9E9, 9E9]];
	VAR robtarget OpenholeUD_1862 := [[497.37, -24.3, 183.82], [0.168821, 0.686658, 0.694077, -0.135121], [0,0,0,0], [9E9, 9E9, 9E9, 9E9, 9E9, 9E9]];
	VAR robtarget OpenholeUD_1863 := [[493.38, -24.3, 183.62], [0.158026, 0.689223, 0.696203, -0.123696], [0,0,0,0], [9E9, 9E9, 9E9, 9E9, 9E9, 9E9]];
	VAR robtarget OpenholeUD_1864 := [[489.38, -24.3, 183.41], [0.146868, 0.691686, 0.698191, -0.111937], [0,0,0,0], [9E9, 9E9, 9E9, 9E9, 9E9, 9E9]];
	VAR robtarget OpenholeUD_1865 := [[485.39, -24.3, 183.21], [0.135356, 0.694031, 0.70002, -0.09986], [0,0,0,0], [9E9, 9E9, 9E9, 9E9, 9E9, 9E9]];
	VAR robtarget OpenholeUD_1866 := [[481.39, -24.3, 183.01], [0.123506, 0.696237, 0.701674, -0.087484], [0,0,0,0], [9E9, 9E9, 9E9, 9E9, 9E9, 9E9]];
	VAR robtarget OpenholeUD_1867 := [[477.4, -24.3, 182.81], [0.111334, 0.698287, 0.703136, -0.074834], [0,0,0,0], [9E9, 9E9, 9E9, 9E9, 9E9, 9E9]];
	VAR robtarget OpenholeUD_1868 := [[473.4, -24.3, 182.6], [0.098863, 0.700161, 0.704389, -0.061939], [0,0,0,0], [9E9, 9E9, 9E9, 9E9, 9E9, 9E9]];
	VAR robtarget OpenholeUD_1869 := [[469.41, -24.3, 182.4], [0.086119, 0.701843, 0.705419, -0.04883], [0,0,0,0], [9E9, 9E9, 9E9, 9E9, 9E9, 9E9]];
	VAR robtarget OpenholeUD_1870 := [[465.41, -24.3, 182.2], [0.073134, 0.703315, 0.706213, -0.035543], [0,0,0,0], [9E9, 9E9, 9E9, 9E9, 9E9, 9E9]];
	VAR robtarget OpenholeUD_1871 := [[461.42, -24.3, 181.99], [0.059941, 0.704562, 0.706761, -0.022119], [0,0,0,0], [9E9, 9E9, 9E9, 9E9, 9E9, 9E9]];
	VAR robtarget OpenholeUD_1872 := [[457.42, -24.3, 181.79], [0.046579, 0.705571, 0.707055, -0.008598], [0,0,0,0], [9E9, 9E9, 9E9, 9E9, 9E9, 9E9]];
	VAR robtarget OpenholeUD_1873 := [[452.65, -24.3, 181.55], [0.03044, 0.706451, 0.707066, 0.007633], [0,0,0,0], [9E9, 9E9, 9E9, 9E9, 9E9, 9E9]];
	VAR robtarget OpenholeUD_1874 := [[452.65, -24.3, 181.55], [0.03044, 0.706451, 0.707066, 0.007633], [0,0,0,0], [9E9, 9E9, 9E9, 9E9, 9E9, 9E9]];
	VAR robtarget OpenholeUD_1875 := [[454.13, -23.1, 181.57], [0.031402, 0.706409, 0.707105, -0.00148], [0,0,0,0], [9E9, 9E9, 9E9, 9E9, 9E9, 9E9]];
	VAR robtarget OpenholeUD_1876 := [[458.13, -23.1, 181.73], [0.044895, 0.70568, 0.706947, -0.015045], [0,0,0,0], [9E9, 9E9, 9E9, 9E9, 9E9, 9E9]];
	VAR robtarget OpenholeUD_1877 := [[462.13, -23.1, 181.88], [0.058259, 0.704703, 0.706531, -0.028541], [0,0,0,0], [9E9, 9E9, 9E9, 9E9, 9E9, 9E9]];
	VAR robtarget OpenholeUD_1878 := [[466.12, -23.1, 182.04], [0.071454, 0.703487, 0.705863, -0.041927], [0,0,0,0], [9E9, 9E9, 9E9, 9E9, 9E9, 9E9]];
	VAR robtarget OpenholeUD_1879 := [[470.12, -23.1, 182.2], [0.084441, 0.702047, 0.704952, -0.05516], [0,0,0,0], [9E9, 9E9, 9E9, 9E9, 9E9, 9E9]];
	VAR robtarget OpenholeUD_1880 := [[474.12, -23.1, 182.35], [0.097187, 0.700396, 0.70381, -0.068202], [0,0,0,0], [9E9, 9E9, 9E9, 9E9, 9E9, 9E9]];
	VAR robtarget OpenholeUD_1881 := [[478.11, -23.1, 182.51], [0.10966, 0.698552, 0.70245, -0.081019], [0,0,0,0], [9E9, 9E9, 9E9, 9E9, 9E9, 9E9]];
	VAR robtarget OpenholeUD_1882 := [[482.11, -23.1, 182.67], [0.121834, 0.696532, 0.700887, -0.09358], [0,0,0,0], [9E9, 9E9, 9E9, 9E9, 9E9, 9E9]];
	VAR robtarget OpenholeUD_1883 := [[486.11, -23.1, 182.82], [0.133687, 0.694354, 0.699138, -0.105857], [0,0,0,0], [9E9, 9E9, 9E9, 9E9, 9E9, 9E9]];
	VAR robtarget OpenholeUD_1884 := [[490.1, -23.1, 182.98], [0.145201, 0.692038, 0.697221, -0.117828], [0,0,0,0], [9E9, 9E9, 9E9, 9E9, 9E9, 9E9]];
	VAR robtarget OpenholeUD_1885 := [[494.1, -23.1, 183.14], [0.156363, 0.689602, 0.695152, -0.129473], [0,0,0,0], [9E9, 9E9, 9E9, 9E9, 9E9, 9E9]];
	VAR robtarget OpenholeUD_1886 := [[498.1, -23.1, 183.29], [0.167162, 0.687064, 0.692951, -0.140777], [0,0,0,0], [9E9, 9E9, 9E9, 9E9, 9E9, 9E9]];
	VAR robtarget OpenholeUD_1887 := [[502.09, -23.1, 183.45], [0.177594, 0.684442, 0.690636, -0.151732], [0,0,0,0], [9E9, 9E9, 9E9, 9E9, 9E9, 9E9]];
	VAR robtarget OpenholeUD_1888 := [[509.35, -23.1, 183.73], [0.183051, 0.683002, 0.683002, -0.183051], [0,0,0,0], [9E9, 9E9, 9E9, 9E9, 9E9, 9E9]];
	VAR robtarget OpenholeUD_1889 := [[513.35, -23.1, 183.72], [0.183051, 0.683002, 0.683002, -0.183051], [0,0,0,0], [9E9, 9E9, 9E9, 9E9, 9E9, 9E9]];
	VAR robtarget OpenholeUD_1890 := [[517.35, -23.1, 183.71], [0.183051, 0.683002, 0.683002, -0.183051], [0,0,0,0], [9E9, 9E9, 9E9, 9E9, 9E9, 9E9]];
	VAR robtarget OpenholeUD_1891 := [[521.35, -23.1, 183.7], [0.183051, 0.683002, 0.683002, -0.183051], [0,0,0,0], [9E9, 9E9, 9E9, 9E9, 9E9, 9E9]];
	VAR robtarget OpenholeUD_1892 := [[529.35, -23.1, 183.67], [0.183051, 0.683002, 0.683002, -0.183051], [0,0,0,0], [9E9, 9E9, 9E9, 9E9, 9E9, 9E9]];
	VAR robtarget OpenholeUD_1893 := [[529.35, -23.1, 183.67], [0.183051, 0.683002, 0.683002, -0.183051], [0,0,0,0], [9E9, 9E9, 9E9, 9E9, 9E9, 9E9]];
	VAR robtarget OpenholeUD_1894 := [[529.35, -21.9, 182.98], [0.183051, 0.683002, 0.683002, -0.183051], [0,0,0,0], [9E9, 9E9, 9E9, 9E9, 9E9, 9E9]];
	VAR robtarget OpenholeUD_1895 := [[525.35, -21.9, 182.99], [0.183051, 0.683002, 0.683002, -0.183051], [0,0,0,0], [9E9, 9E9, 9E9, 9E9, 9E9, 9E9]];
	VAR robtarget OpenholeUD_1896 := [[521.35, -21.9, 183], [0.183051, 0.683002, 0.683002, -0.183051], [0,0,0,0], [9E9, 9E9, 9E9, 9E9, 9E9, 9E9]];
	VAR robtarget OpenholeUD_1897 := [[517.35, -21.9, 183.02], [0.183051, 0.683002, 0.683002, -0.183051], [0,0,0,0], [9E9, 9E9, 9E9, 9E9, 9E9, 9E9]];
	VAR robtarget OpenholeUD_1898 := [[513.35, -21.9, 183.03], [0.183051, 0.683002, 0.683002, -0.183051], [0,0,0,0], [9E9, 9E9, 9E9, 9E9, 9E9, 9E9]];
	VAR robtarget OpenholeUD_1899 := [[509.35, -21.9, 183.04], [0.183051, 0.683002, 0.683002, -0.183051], [0,0,0,0], [9E9, 9E9, 9E9, 9E9, 9E9, 9E9]];
	VAR robtarget OpenholeUD_1900 := [[505.35, -21.9, 182.93], [0.182359, 0.683187, 0.687851, -0.163892], [0,0,0,0], [9E9, 9E9, 9E9, 9E9, 9E9, 9E9]];
	VAR robtarget OpenholeUD_1901 := [[501.35, -21.9, 182.82], [0.172158, 0.685829, 0.690291, -0.153293], [0,0,0,0], [9E9, 9E9, 9E9, 9E9, 9E9, 9E9]];
	VAR robtarget OpenholeUD_1902 := [[497.36, -21.9, 182.71], [0.161586, 0.688397, 0.692633, -0.142335], [0,0,0,0], [9E9, 9E9, 9E9, 9E9, 9E9, 9E9]];
	VAR robtarget OpenholeUD_1903 := [[493.36, -21.9, 182.6], [0.15065, 0.690872, 0.694861, -0.131025], [0,0,0,0], [9E9, 9E9, 9E9, 9E9, 9E9, 9E9]];
	VAR robtarget OpenholeUD_1904 := [[489.36, -21.9, 182.49], [0.139355, 0.693239, 0.696957, -0.119374], [0,0,0,0], [9E9, 9E9, 9E9, 9E9, 9E9, 9E9]];
	VAR robtarget OpenholeUD_1905 := [[485.36, -21.9, 182.38], [0.127712, 0.695478, 0.698903, -0.107398], [0,0,0,0], [9E9, 9E9, 9E9, 9E9, 9E9, 9E9]];
	VAR robtarget OpenholeUD_1906 := [[481.36, -21.9, 182.27], [0.115738, 0.697571, 0.700681, -0.095114], [0,0,0,0], [9E9, 9E9, 9E9, 9E9, 9E9, 9E9]];
	VAR robtarget OpenholeUD_1907 := [[477.36, -21.9, 182.16], [0.10345, 0.699498, 0.702272, -0.082546], [0,0,0,0], [9E9, 9E9, 9E9, 9E9, 9E9, 9E9]];
	VAR robtarget OpenholeUD_1908 := [[473.37, -21.9, 182.05], [0.090873, 0.701243, 0.703661, -0.069722], [0,0,0,0], [9E9, 9E9, 9E9, 9E9, 9E9, 9E9]];
	VAR robtarget OpenholeUD_1909 := [[469.37, -21.9, 181.94], [0.078035, 0.702788, 0.704832, -0.056673], [0,0,0,0], [9E9, 9E9, 9E9, 9E9, 9E9, 9E9]];
	VAR robtarget OpenholeUD_1910 := [[465.37, -21.9, 181.82], [0.064966, 0.704116, 0.705772, -0.043433], [0,0,0,0], [9E9, 9E9, 9E9, 9E9, 9E9, 9E9]];
	VAR robtarget OpenholeUD_1911 := [[461.37, -21.9, 181.71], [0.051703, 0.705214, 0.706468, -0.030043], [0,0,0,0], [9E9, 9E9, 9E9, 9E9, 9E9, 9E9]];
	VAR robtarget OpenholeUD_1912 := [[455, -21.9, 181.54], [0.030286, 0.706458, 0.707056, -0.008515], [0,0,0,0], [9E9, 9E9, 9E9, 9E9, 9E9, 9E9]];
	VAR robtarget OpenholeUD_1913 := [[455, -21.9, 181.54], [0.030286, 0.706458, 0.707056, -0.008515], [0,0,0,0], [9E9, 9E9, 9E9, 9E9, 9E9, 9E9]];
	VAR robtarget OpenholeUD_1914 := [[455.53, -20.7, 181.48], [0.027996, 0.706552, 0.706961, -0.014372], [0,0,0,0], [9E9, 9E9, 9E9, 9E9, 9E9, 9E9]];
	VAR robtarget OpenholeUD_1915 := [[459.53, -20.7, 181.55], [0.041492, 0.705888, 0.706556, -0.027899], [0,0,0,0], [9E9, 9E9, 9E9, 9E9, 9E9, 9E9]];
	VAR robtarget OpenholeUD_1916 := [[463.53, -20.7, 181.61], [0.054858, 0.704976, 0.705898, -0.041328], [0,0,0,0], [9E9, 9E9, 9E9, 9E9, 9E9, 9E9]];
	VAR robtarget OpenholeUD_1917 := [[467.53, -20.7, 181.67], [0.068055, 0.703824, 0.704994, -0.054617], [0,0,0,0], [9E9, 9E9, 9E9, 9E9, 9E9, 9E9]];
	VAR robtarget OpenholeUD_1918 := [[471.53, -20.7, 181.74], [0.081044, 0.702447, 0.703856, -0.067727], [0,0,0,0], [9E9, 9E9, 9E9, 9E9, 9E9, 9E9]];
	VAR robtarget OpenholeUD_1919 := [[475.53, -20.7, 181.8], [0.093791, 0.700859, 0.702496, -0.080621], [0,0,0,0], [9E9, 9E9, 9E9, 9E9, 9E9, 9E9]];
	VAR robtarget OpenholeUD_1920 := [[479.53, -20.7, 181.87], [0.106266, 0.699076, 0.700929, -0.093267], [0,0,0,0], [9E9, 9E9, 9E9, 9E9, 9E9, 9E9]];
	VAR robtarget OpenholeUD_1921 := [[483.53, -20.7, 181.93], [0.118443, 0.697116, 0.699172, -0.105636], [0,0,0,0], [9E9, 9E9, 9E9, 9E9, 9E9, 9E9]];
	VAR robtarget OpenholeUD_1922 := [[487.53, -20.7, 182], [0.1303, 0.694998, 0.697242, -0.117704], [0,0,0,0], [9E9, 9E9, 9E9, 9E9, 9E9, 9E9]];
	VAR robtarget OpenholeUD_1923 := [[491.53, -20.7, 182.06], [0.14182, 0.692739, 0.695157, -0.12945], [0,0,0,0], [9E9, 9E9, 9E9, 9E9, 9E9, 9E9]];
	VAR robtarget OpenholeUD_1924 := [[495.53, -20.7, 182.13], [0.152989, 0.690358, 0.692935, -0.140858], [0,0,0,0], [9E9, 9E9, 9E9, 9E9, 9E9, 9E9]];
	VAR robtarget OpenholeUD_1925 := [[499.53, -20.7, 182.19], [0.163797, 0.687874, 0.690595, -0.151916], [0,0,0,0], [9E9, 9E9, 9E9, 9E9, 9E9, 9E9]];
	VAR robtarget OpenholeUD_1926 := [[503.53, -20.7, 182.25], [0.174239, 0.685303, 0.688154, -0.162616], [0,0,0,0], [9E9, 9E9, 9E9, 9E9, 9E9, 9E9]];
	VAR robtarget OpenholeUD_1927 := [[509.35, -20.7, 182.35], [0.183051, 0.683002, 0.683002, -0.183051], [0,0,0,0], [9E9, 9E9, 9E9, 9E9, 9E9, 9E9]];
	VAR robtarget OpenholeUD_1928 := [[513.35, -20.7, 182.34], [0.183051, 0.683002, 0.683002, -0.183051], [0,0,0,0], [9E9, 9E9, 9E9, 9E9, 9E9, 9E9]];
	VAR robtarget OpenholeUD_1929 := [[517.35, -20.7, 182.32], [0.183051, 0.683002, 0.683002, -0.183051], [0,0,0,0], [9E9, 9E9, 9E9, 9E9, 9E9, 9E9]];
	VAR robtarget OpenholeUD_1930 := [[521.35, -20.7, 182.31], [0.183051, 0.683002, 0.683002, -0.183051], [0,0,0,0], [9E9, 9E9, 9E9, 9E9, 9E9, 9E9]];
	VAR robtarget OpenholeUD_1931 := [[525.35, -20.7, 182.3], [0.183051, 0.683002, 0.683002, -0.183051], [0,0,0,0], [9E9, 9E9, 9E9, 9E9, 9E9, 9E9]];
	VAR robtarget OpenholeUD_1932 := [[529.35, -20.7, 182.29], [0.183051, 0.683002, 0.683002, -0.183051], [0,0,0,0], [9E9, 9E9, 9E9, 9E9, 9E9, 9E9]];
	VAR robtarget OpenholeUD_1933 := [[529.35, -20.7, 182.29], [0.183051, 0.683002, 0.683002, -0.183051], [0,0,0,0], [9E9, 9E9, 9E9, 9E9, 9E9, 9E9]];
	VAR robtarget OpenholeUD_1934 := [[529.35, -19.5, 181.59], [0.183051, 0.683002, 0.683002, -0.183051], [0,0,0,0], [9E9, 9E9, 9E9, 9E9, 9E9, 9E9]];
	VAR robtarget OpenholeUD_1935 := [[525.35, -19.5, 181.6], [0.183051, 0.683002, 0.683002, -0.183051], [0,0,0,0], [9E9, 9E9, 9E9, 9E9, 9E9, 9E9]];
	VAR robtarget OpenholeUD_1936 := [[521.35, -19.5, 181.62], [0.183051, 0.683002, 0.683002, -0.183051], [0,0,0,0], [9E9, 9E9, 9E9, 9E9, 9E9, 9E9]];
	VAR robtarget OpenholeUD_1937 := [[517.35, -19.5, 181.63], [0.183051, 0.683002, 0.683002, -0.183051], [0,0,0,0], [9E9, 9E9, 9E9, 9E9, 9E9, 9E9]];
	VAR robtarget OpenholeUD_1938 := [[513.35, -19.5, 181.64], [0.183051, 0.683002, 0.683002, -0.183051], [0,0,0,0], [9E9, 9E9, 9E9, 9E9, 9E9, 9E9]];
	VAR robtarget OpenholeUD_1939 := [[509.35, -19.5, 181.65], [0.183051, 0.683002, 0.683002, -0.183051], [0,0,0,0], [9E9, 9E9, 9E9, 9E9, 9E9, 9E9]];
	VAR robtarget OpenholeUD_1940 := [[505.35, -19.5, 181.64], [0.175396, 0.685008, 0.686154, -0.170859], [0,0,0,0], [9E9, 9E9, 9E9, 9E9, 9E9, 9E9]];
	VAR robtarget OpenholeUD_1941 := [[501.35, -19.5, 181.62], [0.165053, 0.687574, 0.688676, -0.160392], [0,0,0,0], [9E9, 9E9, 9E9, 9E9, 9E9, 9E9]];
	VAR robtarget OpenholeUD_1942 := [[497.35, -19.5, 181.6], [0.154342, 0.690057, 0.691109, -0.149561], [0,0,0,0], [9E9, 9E9, 9E9, 9E9, 9E9, 9E9]];
	VAR robtarget OpenholeUD_1943 := [[493.35, -19.5, 181.58], [0.14327, 0.69244, 0.693435, -0.138374], [0,0,0,0], [9E9, 9E9, 9E9, 9E9, 9E9, 9E9]];
	VAR robtarget OpenholeUD_1944 := [[489.35, -19.5, 181.56], [0.131845, 0.694706, 0.695638, -0.12684], [0,0,0,0], [9E9, 9E9, 9E9, 9E9, 9E9, 9E9]];
	VAR robtarget OpenholeUD_1945 := [[485.35, -19.5, 181.55], [0.12008, 0.696836, 0.697697, -0.114972], [0,0,0,0], [9E9, 9E9, 9E9, 9E9, 9E9, 9E9]];
	VAR robtarget OpenholeUD_1946 := [[481.35, -19.5, 181.53], [0.107989, 0.698812, 0.699596, -0.102789], [0,0,0,0], [9E9, 9E9, 9E9, 9E9, 9E9, 9E9]];
	VAR robtarget OpenholeUD_1947 := [[477.35, -19.5, 181.51], [0.095595, 0.700615, 0.701316, -0.090313], [0,0,0,0], [9E9, 9E9, 9E9, 9E9, 9E9, 9E9]];
	VAR robtarget OpenholeUD_1948 := [[473.35, -19.5, 181.49], [0.082921, 0.702228, 0.702839, -0.07757], [0,0,0,0], [9E9, 9E9, 9E9, 9E9, 9E9, 9E9]];
	VAR robtarget OpenholeUD_1949 := [[469.35, -19.5, 181.47], [0.069996, 0.703634, 0.704151, -0.06459], [0,0,0,0], [9E9, 9E9, 9E9, 9E9, 9E9, 9E9]];
	VAR robtarget OpenholeUD_1950 := [[465.35, -19.5, 181.45], [0.056854, 0.704817, 0.705236, -0.051408], [0,0,0,0], [9E9, 9E9, 9E9, 9E9, 9E9, 9E9]];
	VAR robtarget OpenholeUD_1951 := [[461.35, -19.5, 181.44], [0.043532, 0.705766, 0.706082, -0.03806], [0,0,0,0], [9E9, 9E9, 9E9, 9E9, 9E9, 9E9]];
	VAR robtarget OpenholeUD_1952 := [[455.8, -19.5, 181.41], [0.024819, 0.706671, 0.706842, -0.019341], [0,0,0,0], [9E9, 9E9, 9E9, 9E9, 9E9, 9E9]];
	VAR robtarget OpenholeUD_1953 := [[455.8, -19.5, 181.41], [0.024819, 0.706671, 0.706842, -0.019341], [0,0,0,0], [9E9, 9E9, 9E9, 9E9, 9E9, 9E9]];
	VAR robtarget OpenholeUD_1954 := [[455.83, -18.3, 181.34], [0.020866, 0.706799, 0.706715, -0.023535], [0,0,0,0], [9E9, 9E9, 9E9, 9E9, 9E9, 9E9]];
	VAR robtarget OpenholeUD_1955 := [[459.83, -18.3, 181.31], [0.034389, 0.70627, 0.706137, -0.037027], [0,0,0,0], [9E9, 9E9, 9E9, 9E9, 9E9, 9E9]];
	VAR robtarget OpenholeUD_1956 := [[463.83, -18.3, 181.28], [0.047793, 0.70549, 0.705308, -0.050403], [0,0,0,0], [9E9, 9E9, 9E9, 9E9, 9E9, 9E9]];
	VAR robtarget OpenholeUD_1957 := [[467.83, -18.3, 181.25], [0.061038, 0.704467, 0.704239, -0.063623], [0,0,0,0], [9E9, 9E9, 9E9, 9E9, 9E9, 9E9]];
	VAR robtarget OpenholeUD_1958 := [[471.83, -18.3, 181.22], [0.074086, 0.703215, 0.70294, -0.076648], [0,0,0,0], [9E9, 9E9, 9E9, 9E9, 9E9, 9E9]];
	VAR robtarget OpenholeUD_1959 := [[475.83, -18.3, 181.2], [0.086901, 0.701747, 0.701427, -0.089442], [0,0,0,0], [9E9, 9E9, 9E9, 9E9, 9E9, 9E9]];
	VAR robtarget OpenholeUD_1960 := [[479.83, -18.3, 181.17], [0.099453, 0.700078, 0.699715, -0.101976], [0,0,0,0], [9E9, 9E9, 9E9, 9E9, 9E9, 9E9]];
	VAR robtarget OpenholeUD_1961 := [[483.83, -18.3, 181.14], [0.111714, 0.698226, 0.697821, -0.11422], [0,0,0,0], [9E9, 9E9, 9E9, 9E9, 9E9, 9E9]];
	VAR robtarget OpenholeUD_1962 := [[487.83, -18.3, 181.11], [0.123662, 0.69621, 0.695763, -0.126152], [0,0,0,0], [9E9, 9E9, 9E9, 9E9, 9E9, 9E9]];
	VAR robtarget OpenholeUD_1963 := [[491.83, -18.3, 181.08], [0.135278, 0.694046, 0.693559, -0.137755], [0,0,0,0], [9E9, 9E9, 9E9, 9E9, 9E9, 9E9]];
	VAR robtarget OpenholeUD_1964 := [[495.83, -18.3, 181.06], [0.146549, 0.691754, 0.691228, -0.149011], [0,0,0,0], [9E9, 9E9, 9E9, 9E9, 9E9, 9E9]];
	VAR robtarget OpenholeUD_1965 := [[499.83, -18.3, 181.03], [0.157463, 0.689351, 0.688787, -0.159912], [0,0,0,0], [9E9, 9E9, 9E9, 9E9, 9E9, 9E9]];
	VAR robtarget OpenholeUD_1966 := [[503.83, -18.3, 181], [0.168014, 0.686856, 0.686256, -0.17045], [0,0,0,0], [9E9, 9E9, 9E9, 9E9, 9E9, 9E9]];
	VAR robtarget OpenholeUD_1967 := [[509.35, -18.3, 180.96], [0.183051, 0.683002, 0.683002, -0.183051], [0,0,0,0], [9E9, 9E9, 9E9, 9E9, 9E9, 9E9]];
	VAR robtarget OpenholeUD_1968 := [[513.35, -18.3, 180.95], [0.183051, 0.683002, 0.683002, -0.183051], [0,0,0,0], [9E9, 9E9, 9E9, 9E9, 9E9, 9E9]];
	VAR robtarget OpenholeUD_1969 := [[517.35, -18.3, 180.94], [0.183051, 0.683002, 0.683002, -0.183051], [0,0,0,0], [9E9, 9E9, 9E9, 9E9, 9E9, 9E9]];
	VAR robtarget OpenholeUD_1970 := [[521.35, -18.3, 180.92], [0.183051, 0.683002, 0.683002, -0.183051], [0,0,0,0], [9E9, 9E9, 9E9, 9E9, 9E9, 9E9]];
	VAR robtarget OpenholeUD_1971 := [[525.35, -18.3, 180.91], [0.183051, 0.683002, 0.683002, -0.183051], [0,0,0,0], [9E9, 9E9, 9E9, 9E9, 9E9, 9E9]];
	VAR robtarget OpenholeUD_1972 := [[529.35, -18.3, 180.9], [0.183051, 0.683002, 0.683002, -0.183051], [0,0,0,0], [9E9, 9E9, 9E9, 9E9, 9E9, 9E9]];
	VAR robtarget OpenholeUD_1973 := [[529.35, -18.3, 180.9], [0.183051, 0.683002, 0.683002, -0.183051], [0,0,0,0], [9E9, 9E9, 9E9, 9E9, 9E9, 9E9]];
	VAR robtarget OpenholeUD_1974 := [[529.34, -17.1, 180.21], [0.183051, 0.683002, 0.683002, -0.183051], [0,0,0,0], [9E9, 9E9, 9E9, 9E9, 9E9, 9E9]];
	VAR robtarget OpenholeUD_1975 := [[525.34, -17.1, 180.22], [0.183051, 0.683002, 0.683002, -0.183051], [0,0,0,0], [9E9, 9E9, 9E9, 9E9, 9E9, 9E9]];
	VAR robtarget OpenholeUD_1976 := [[521.34, -17.1, 180.23], [0.183051, 0.683002, 0.683002, -0.183051], [0,0,0,0], [9E9, 9E9, 9E9, 9E9, 9E9, 9E9]];
	VAR robtarget OpenholeUD_1977 := [[517.34, -17.1, 180.24], [0.183051, 0.683002, 0.683002, -0.183051], [0,0,0,0], [9E9, 9E9, 9E9, 9E9, 9E9, 9E9]];
	VAR robtarget OpenholeUD_1978 := [[513.34, -17.1, 180.26], [0.183051, 0.683002, 0.683002, -0.183051], [0,0,0,0], [9E9, 9E9, 9E9, 9E9, 9E9, 9E9]];
	VAR robtarget OpenholeUD_1979 := [[509.34, -17.1, 180.27], [0.183051, 0.683002, 0.683002, -0.183051], [0,0,0,0], [9E9, 9E9, 9E9, 9E9, 9E9, 9E9]];
	VAR robtarget OpenholeUD_1980 := [[505.34, -17.1, 180.34], [0.168418, 0.686757, 0.684384, -0.177816], [0,0,0,0], [9E9, 9E9, 9E9, 9E9, 9E9, 9E9]];
	VAR robtarget OpenholeUD_1981 := [[501.34, -17.1, 180.42], [0.157938, 0.689243, 0.686985, -0.167487], [0,0,0,0], [9E9, 9E9, 9E9, 9E9, 9E9, 9E9]];
	VAR robtarget OpenholeUD_1982 := [[497.35, -17.1, 180.49], [0.147096, 0.691638, 0.689505, -0.156791], [0,0,0,0], [9E9, 9E9, 9E9, 9E9, 9E9, 9E9]];
	VAR robtarget OpenholeUD_1983 := [[493.35, -17.1, 180.57], [0.135896, 0.693925, 0.691926, -0.145734], [0,0,0,0], [9E9, 9E9, 9E9, 9E9, 9E9, 9E9]];
	VAR robtarget OpenholeUD_1984 := [[489.35, -17.1, 180.64], [0.124349, 0.696087, 0.694231, -0.134324], [0,0,0,0], [9E9, 9E9, 9E9, 9E9, 9E9, 9E9]];
	VAR robtarget OpenholeUD_1985 := [[485.35, -17.1, 180.71], [0.112468, 0.698105, 0.696402, -0.122574], [0,0,0,0], [9E9, 9E9, 9E9, 9E9, 9E9, 9E9]];
	VAR robtarget OpenholeUD_1986 := [[481.35, -17.1, 180.79], [0.10027, 0.699961, 0.698419, -0.110501], [0,0,0,0], [9E9, 9E9, 9E9, 9E9, 9E9, 9E9]];
	VAR robtarget OpenholeUD_1987 := [[477.35, -17.1, 180.86], [0.087777, 0.701637, 0.700265, -0.098126], [0,0,0,0], [9E9, 9E9, 9E9, 9E9, 9E9, 9E9]];
	VAR robtarget OpenholeUD_1988 := [[473.35, -17.1, 180.94], [0.075016, 0.703116, 0.701922, -0.085473], [0,0,0,0], [9E9, 9E9, 9E9, 9E9, 9E9, 9E9]];
	VAR robtarget OpenholeUD_1989 := [[469.35, -17.1, 181.01], [0.062015, 0.704382, 0.703373, -0.072572], [0,0,0,0], [9E9, 9E9, 9E9, 9E9, 9E9, 9E9]];
	VAR robtarget OpenholeUD_1990 := [[465.35, -17.1, 181.08], [0.04881, 0.70542, 0.704603, -0.059456], [0,0,0,0], [9E9, 9E9, 9E9, 9E9, 9E9, 9E9]];
	VAR robtarget OpenholeUD_1991 := [[461.35, -17.1, 181.16], [0.035437, 0.706218, 0.705598, -0.046162], [0,0,0,0], [9E9, 9E9, 9E9, 9E9, 9E9, 9E9]];
	VAR robtarget OpenholeUD_1992 := [[455.65, -17.1, 181.26], [0.01615, 0.706922, 0.706592, -0.026967], [0,0,0,0], [9E9, 9E9, 9E9, 9E9, 9E9, 9E9]];
	VAR robtarget OpenholeUD_1993 := [[455.65, -17.1, 181.26], [0.01615, 0.706922, 0.706592, -0.026967], [0,0,0,0], [9E9, 9E9, 9E9, 9E9, 9E9, 9E9]];
	VAR robtarget OpenholeUD_1994 := [[455.21, -15.9, 181.2], [0.010597, 0.707027, 0.706488, -0.029566], [0,0,0,0], [9E9, 9E9, 9E9, 9E9, 9E9, 9E9]];
	VAR robtarget OpenholeUD_1995 := [[459.21, -15.9, 181.08], [0.024158, 0.706694, 0.705796, -0.043037], [0,0,0,0], [9E9, 9E9, 9E9, 9E9, 9E9, 9E9]];
	VAR robtarget OpenholeUD_1996 := [[463.21, -15.9, 180.96], [0.037622, 0.706105, 0.704855, -0.056384], [0,0,0,0], [9E9, 9E9, 9E9, 9E9, 9E9, 9E9]];
	VAR robtarget OpenholeUD_1997 := [[467.21, -15.9, 180.84], [0.050947, 0.705269, 0.703676, -0.069568], [0,0,0,0], [9E9, 9E9, 9E9, 9E9, 9E9, 9E9]];
	VAR robtarget OpenholeUD_1998 := [[471.2, -15.9, 180.72], [0.064093, 0.704196, 0.702272, -0.082549], [0,0,0,0], [9E9, 9E9, 9E9, 9E9, 9E9, 9E9]];
	VAR robtarget OpenholeUD_1999 := [[475.2, -15.9, 180.6], [0.077025, 0.702899, 0.700656, -0.095294], [0,0,0,0], [9E9, 9E9, 9E9, 9E9, 9E9, 9E9]];
	VAR robtarget OpenholeUD_2000 := [[479.2, -15.9, 180.48], [0.089708, 0.701393, 0.698846, -0.107771], [0,0,0,0], [9E9, 9E9, 9E9, 9E9, 9E9, 9E9]];
	VAR robtarget OpenholeUD_2001 := [[483.2, -15.9, 180.36], [0.102116, 0.699694, 0.696858, -0.119954], [0,0,0,0], [9E9, 9E9, 9E9, 9E9, 9E9, 9E9]];
	VAR robtarget OpenholeUD_2002 := [[487.2, -15.9, 180.24], [0.114222, 0.69782, 0.694711, -0.13182], [0,0,0,0], [9E9, 9E9, 9E9, 9E9, 9E9, 9E9]];
	VAR robtarget OpenholeUD_2003 := [[491.2, -15.9, 180.12], [0.126007, 0.695789, 0.692424, -0.143351], [0,0,0,0], [9E9, 9E9, 9E9, 9E9, 9E9, 9E9]];
	VAR robtarget OpenholeUD_2004 := [[495.19, -15.9, 180], [0.137455, 0.693618, 0.690014, -0.154533], [0,0,0,0], [9E9, 9E9, 9E9, 9E9, 9E9, 9E9]];
	VAR robtarget OpenholeUD_2005 := [[499.19, -15.9, 179.88], [0.148553, 0.691326, 0.687501, -0.165355], [0,0,0,0], [9E9, 9E9, 9E9, 9E9, 9E9, 9E9]];
	VAR robtarget OpenholeUD_2006 := [[503.19, -15.9, 179.76], [0.159293, 0.688931, 0.684902, -0.175812], [0,0,0,0], [9E9, 9E9, 9E9, 9E9, 9E9, 9E9]];
	VAR robtarget OpenholeUD_2007 := [[509.34, -15.9, 179.58], [0.183051, 0.683002, 0.683002, -0.183051], [0,0,0,0], [9E9, 9E9, 9E9, 9E9, 9E9, 9E9]];
	VAR robtarget OpenholeUD_2008 := [[513.34, -15.9, 179.56], [0.183051, 0.683002, 0.683002, -0.183051], [0,0,0,0], [9E9, 9E9, 9E9, 9E9, 9E9, 9E9]];
	VAR robtarget OpenholeUD_2009 := [[517.34, -15.9, 179.55], [0.183051, 0.683002, 0.683002, -0.183051], [0,0,0,0], [9E9, 9E9, 9E9, 9E9, 9E9, 9E9]];
	VAR robtarget OpenholeUD_2010 := [[521.34, -15.9, 179.54], [0.183051, 0.683002, 0.683002, -0.183051], [0,0,0,0], [9E9, 9E9, 9E9, 9E9, 9E9, 9E9]];
	VAR robtarget OpenholeUD_2011 := [[525.34, -15.9, 179.53], [0.183051, 0.683002, 0.683002, -0.183051], [0,0,0,0], [9E9, 9E9, 9E9, 9E9, 9E9, 9E9]];
	VAR robtarget OpenholeUD_2012 := [[529.34, -15.9, 179.51], [0.183051, 0.683002, 0.683002, -0.183051], [0,0,0,0], [9E9, 9E9, 9E9, 9E9, 9E9, 9E9]];
	VAR robtarget OpenholeUD_2013 := [[529.34, -15.9, 179.51], [0.183051, 0.683002, 0.683002, -0.183051], [0,0,0,0], [9E9, 9E9, 9E9, 9E9, 9E9, 9E9]];
	VAR robtarget OpenholeUD_2014 := [[529.34, -14.7, 178.82], [0.183051, 0.683002, 0.683002, -0.183051], [0,0,0,0], [9E9, 9E9, 9E9, 9E9, 9E9, 9E9]];
	VAR robtarget OpenholeUD_2015 := [[525.34, -14.7, 178.83], [0.183051, 0.683002, 0.683002, -0.183051], [0,0,0,0], [9E9, 9E9, 9E9, 9E9, 9E9, 9E9]];
	VAR robtarget OpenholeUD_2016 := [[521.34, -14.7, 178.85], [0.183051, 0.683002, 0.683002, -0.183051], [0,0,0,0], [9E9, 9E9, 9E9, 9E9, 9E9, 9E9]];
	VAR robtarget OpenholeUD_2017 := [[517.34, -14.7, 178.86], [0.183051, 0.683002, 0.683002, -0.183051], [0,0,0,0], [9E9, 9E9, 9E9, 9E9, 9E9, 9E9]];
	VAR robtarget OpenholeUD_2018 := [[513.34, -14.7, 178.87], [0.183051, 0.683002, 0.683002, -0.183051], [0,0,0,0], [9E9, 9E9, 9E9, 9E9, 9E9, 9E9]];
	VAR robtarget OpenholeUD_2019 := [[509.34, -14.7, 178.88], [0.183051, 0.683002, 0.683002, -0.183051], [0,0,0,0], [9E9, 9E9, 9E9, 9E9, 9E9, 9E9]];
	VAR robtarget OpenholeUD_2020 := [[505.34, -14.7, 179.05], [0.161432, 0.688433, 0.682543, -0.184757], [0,0,0,0], [9E9, 9E9, 9E9, 9E9, 9E9, 9E9]];
	VAR robtarget OpenholeUD_2021 := [[501.35, -14.7, 179.22], [0.150823, 0.690835, 0.685219, -0.174571], [0,0,0,0], [9E9, 9E9, 9E9, 9E9, 9E9, 9E9]];
	VAR robtarget OpenholeUD_2022 := [[497.35, -14.7, 179.38], [0.139855, 0.693138, 0.687822, -0.164016], [0,0,0,0], [9E9, 9E9, 9E9, 9E9, 9E9, 9E9]];
	VAR robtarget OpenholeUD_2023 := [[493.35, -14.7, 179.55], [0.128535, 0.695326, 0.690334, -0.153096], [0,0,0,0], [9E9, 9E9, 9E9, 9E9, 9E9, 9E9]];
	VAR robtarget OpenholeUD_2024 := [[489.36, -14.7, 179.72], [0.116874, 0.697381, 0.692739, -0.141819], [0,0,0,0], [9E9, 9E9, 9E9, 9E9, 9E9, 9E9]];
	VAR robtarget OpenholeUD_2025 := [[485.36, -14.7, 179.88], [0.104886, 0.699285, 0.695017, -0.130195], [0,0,0,0], [9E9, 9E9, 9E9, 9E9, 9E9, 9E9]];
	VAR robtarget OpenholeUD_2026 := [[481.36, -14.7, 180.05], [0.09259, 0.701019, 0.697151, -0.11824], [0,0,0,0], [9E9, 9E9, 9E9, 9E9, 9E9, 9E9]];
	VAR robtarget OpenholeUD_2027 := [[477.37, -14.7, 180.21], [0.080008, 0.702566, 0.69912, -0.105974], [0,0,0,0], [9E9, 9E9, 9E9, 9E9, 9E9, 9E9]];
	VAR robtarget OpenholeUD_2028 := [[473.37, -14.7, 180.38], [0.067168, 0.703909, 0.700908, -0.093421], [0,0,0,0], [9E9, 9E9, 9E9, 9E9, 9E9, 9E9]];
	VAR robtarget OpenholeUD_2029 := [[469.37, -14.7, 180.55], [0.054102, 0.705034, 0.702497, -0.080608], [0,0,0,0], [9E9, 9E9, 9E9, 9E9, 9E9, 9E9]];
	VAR robtarget OpenholeUD_2030 := [[465.38, -14.7, 180.71], [0.040842, 0.705926, 0.703871, -0.067568], [0,0,0,0], [9E9, 9E9, 9E9, 9E9, 9E9, 9E9]];
	VAR robtarget OpenholeUD_2031 := [[461.38, -14.7, 180.88], [0.027429, 0.706575, 0.705016, -0.054337], [0,0,0,0], [9E9, 9E9, 9E9, 9E9, 9E9, 9E9]];
	VAR robtarget OpenholeUD_2032 := [[454.47, -14.7, 181.17], [0.003993, 0.707096, 0.706422, -0.03112], [0,0,0,0], [9E9, 9E9, 9E9, 9E9, 9E9, 9E9]];
	VAR robtarget OpenholeUD_2033 := [[454.47, -14.7, 181.17], [0.003993, 0.707096, 0.706422, -0.03112], [0,0,0,0], [9E9, 9E9, 9E9, 9E9, 9E9, 9E9]];
	VAR robtarget OpenholeUD_2034 := [[453.25, -13.5, 181.17], [-0.00425, 0.707094, 0.706425, -0.031044], [0,0,0,0], [9E9, 9E9, 9E9, 9E9, 9E9, 9E9]];
	VAR robtarget OpenholeUD_2035 := [[457.24, -13.5, 180.96], [0.009349, 0.707045, 0.705704, -0.044523], [0,0,0,0], [9E9, 9E9, 9E9, 9E9, 9E9, 9E9]];
	VAR robtarget OpenholeUD_2036 := [[461.24, -13.5, 180.75], [0.022888, 0.706736, 0.704734, -0.057885], [0,0,0,0], [9E9, 9E9, 9E9, 9E9, 9E9, 9E9]];
	VAR robtarget OpenholeUD_2037 := [[465.23, -13.5, 180.54], [0.036324, 0.706173, 0.703524, -0.071089], [0,0,0,0], [9E9, 9E9, 9E9, 9E9, 9E9, 9E9]];
	VAR robtarget OpenholeUD_2038 := [[469.22, -13.5, 180.32], [0.049613, 0.705364, 0.702088, -0.084097], [0,0,0,0], [9E9, 9E9, 9E9, 9E9, 9E9, 9E9]];
	VAR robtarget OpenholeUD_2039 := [[473.22, -13.5, 180.11], [0.062718, 0.70432, 0.70044, -0.096872], [0,0,0,0], [9E9, 9E9, 9E9, 9E9, 9E9, 9E9]];
	VAR robtarget OpenholeUD_2040 := [[477.21, -13.5, 179.9], [0.075603, 0.703053, 0.698595, -0.109384], [0,0,0,0], [9E9, 9E9, 9E9, 9E9, 9E9, 9E9]];
	VAR robtarget OpenholeUD_2041 := [[481.21, -13.5, 179.69], [0.088237, 0.70158, 0.696572, -0.121605], [0,0,0,0], [9E9, 9E9, 9E9, 9E9, 9E9, 9E9]];
	VAR robtarget OpenholeUD_2042 := [[485.2, -13.5, 179.47], [0.100591, 0.699915, 0.694388, -0.133511], [0,0,0,0], [9E9, 9E9, 9E9, 9E9, 9E9, 9E9]];
	VAR robtarget OpenholeUD_2043 := [[489.2, -13.5, 179.26], [0.112642, 0.698077, 0.692063, -0.145084], [0,0,0,0], [9E9, 9E9, 9E9, 9E9, 9E9, 9E9]];
	VAR robtarget OpenholeUD_2044 := [[493.19, -13.5, 179.05], [0.124372, 0.696083, 0.689614, -0.156308], [0,0,0,0], [9E9, 9E9, 9E9, 9E9, 9E9, 9E9]];
	VAR robtarget OpenholeUD_2045 := [[497.18, -13.5, 178.84], [0.135763, 0.693951, 0.687061, -0.167172], [0,0,0,0], [9E9, 9E9, 9E9, 9E9, 9E9, 9E9]];
	VAR robtarget OpenholeUD_2046 := [[501.18, -13.5, 178.62], [0.146806, 0.691699, 0.684422, -0.17767], [0,0,0,0], [9E9, 9E9, 9E9, 9E9, 9E9, 9E9]];
	VAR robtarget OpenholeUD_2047 := [[505.17, -13.5, 178.41], [0.157492, 0.689345, 0.681713, -0.187797], [0,0,0,0], [9E9, 9E9, 9E9, 9E9, 9E9, 9E9]];
	VAR robtarget OpenholeUD_2048 := [[509.34, -13.5, 178.19], [0.183051, 0.683002, 0.683002, -0.183051], [0,0,0,0], [9E9, 9E9, 9E9, 9E9, 9E9, 9E9]];
	VAR robtarget OpenholeUD_2049 := [[513.34, -13.5, 178.18], [0.183051, 0.683002, 0.683002, -0.183051], [0,0,0,0], [9E9, 9E9, 9E9, 9E9, 9E9, 9E9]];
	VAR robtarget OpenholeUD_2050 := [[517.34, -13.5, 178.16], [0.183051, 0.683002, 0.683002, -0.183051], [0,0,0,0], [9E9, 9E9, 9E9, 9E9, 9E9, 9E9]];
	VAR robtarget OpenholeUD_2051 := [[521.34, -13.5, 178.15], [0.183051, 0.683002, 0.683002, -0.183051], [0,0,0,0], [9E9, 9E9, 9E9, 9E9, 9E9, 9E9]];
	VAR robtarget OpenholeUD_2052 := [[529.34, -13.5, 178.13], [0.183051, 0.683002, 0.683002, -0.183051], [0,0,0,0], [9E9, 9E9, 9E9, 9E9, 9E9, 9E9]];
	VAR robtarget OpenholeUD_2053 := [[529.34, -13.5, 178.13], [0.183051, 0.683002, 0.683002, -0.183051], [0,0,0,0], [9E9, 9E9, 9E9, 9E9, 9E9, 9E9]];
	VAR robtarget OpenholeUD_2054 := [[529.33, -12.3, 177.43], [0.183051, 0.683002, 0.683002, -0.183051], [0,0,0,0], [9E9, 9E9, 9E9, 9E9, 9E9, 9E9]];
	VAR robtarget OpenholeUD_2055 := [[525.33, -12.3, 177.45], [0.183051, 0.683002, 0.683002, -0.183051], [0,0,0,0], [9E9, 9E9, 9E9, 9E9, 9E9, 9E9]];
	VAR robtarget OpenholeUD_2056 := [[521.33, -12.3, 177.46], [0.183051, 0.683002, 0.683002, -0.183051], [0,0,0,0], [9E9, 9E9, 9E9, 9E9, 9E9, 9E9]];
	VAR robtarget OpenholeUD_2057 := [[517.33, -12.3, 177.47], [0.183051, 0.683002, 0.683002, -0.183051], [0,0,0,0], [9E9, 9E9, 9E9, 9E9, 9E9, 9E9]];
